// SIMATIC STEP 7 (V5.x) project KROMOSS_RULLIERA_EIDOS
// station: Hardware
// station: SIMATIC 300
// station: P_ADR_BUS
// station: P_ADR_BUS
// station: Configurazione
// program: Programma S7
// program: Backup
// program: MICROMASTER_420
// program: MICROMASTER_420
// program: MICROMASTER_420
// program: MICROMASTER_420
// program: MICROMASTER_420
// program: MICROMASTER_420
// program: MICROMASTER_420
// program: MICROMASTER_420
// program: MICROMASTER_420
// program: MICROMASTER_420
// program: MICROMASTER_420
// program: MICROMASTER_420
// program: MICROMASTER_420
// program: MICROMASTER_420
// program: MICROMASTER_420
// program: MICROMASTER_420

SYMBOL_TABLE
"C1"	C 1	COUNTER	// TIMEOUT TRASFERIMENTO "M3"
"C2"	C 2	COUNTER	// TEMPO SVUOTAMENTO CATENA INGRESSO CADENZATORE LINEA 2
"C3"	C 3	COUNTER	// TEMPO PASSO CATENE LINEA 2
"C4"	C 4	COUNTER	// TEMPO PASSO CATENE ACCUMULO "A" LINEA 2
"C5"	C 5	COUNTER	// TEMPO SVUOTAMENTO CATENA INGRESSO CADENZATORE LINEA 1
"C6"	C 6	COUNTER	// TEMPO PASSO CATENE LINEA 1
"C7"	C 7	COUNTER
"C8"	C 8	COUNTER
"C9"	C 9	COUNTER	// CONTEGGIO PEZZI SU CATENA FISSA LINEA 2
"C10"	C 10	COUNTER
"C11"	C 11	COUNTER
"C12"	C 12	COUNTER
"C13"	C 13	COUNTER	// CONTEGGIO PEZZI SU CATENA FISSA LINEA 1
"C14"	C 14	COUNTER
"C15"	C 15	COUNTER
"C16"	C 16	COUNTER
"C17"	C 17	COUNTER
"C18"	C 18	COUNTER
"C19"	C 19	COUNTER
"C20"	C 20	COUNTER	// RITARDO FUORI INGOMBRO M22
"C21"	C 21	COUNTER	// RITARDO FUORI INGOMBRO M24
"DB_OP"	DB 2	DB 2
"DB_InverterParams"	DB 3	DB 3
"DB_Accumulo"	DB 10	DB 10
"DETAIL_DIAG_DB"	DB 125	FB 125
"DB_ReadParamLoop"	DB 211	FB 211
"DB_GestCodeEstrusori"	DB 212	FB 212
"DB_LinkEthernet_1"	DB 213	FB 213
"DB_LinkEthernet_2"	DB 214	FB 213
"DETAIL_DP_DIAG"	FB 125	FB 125
"ReadParamInverters"	FB 210	FB 210
"FB_ReadParamLoop"	FB 211	FB 211
"FB_GestCodeEstrusori"	FB 212	FB 212
"FB_LinkEthernet"	FB 213	FB 213
"Allarmi"	FC 1	FC 1	// Gestione allarmi
"Segnalazioni"	FC 2	FC 2	// Gestione segnalazioni
"Consensi Generali"	FC 3	FC 3	// Consensi generali
"Automatico_zona_ingresso"	FC 4	FC 4	// Condizioni automatico zona ingresso
"Automatico_linea_1"	FC 5	FC 5	// Condizioni automatico linea 1
"Automatico_linea_2"	FC 6	FC 6	// Condizioni automatico linea 2
"PROFIBUS_MM4"	FC 10	FC 10
"Comandi_zona_ingresso"	FC 14	FC 14	// Comandi utenze zona ingresso
"Comandi_linea_1"	FC 15	FC 15	// Comandi utenze linea 1
"Comandi_linea_2"	FC 16	FC 16	// Comandi utenze linea 2
"Comandi_Inverter"	FC 17	FC 17
"Gestione finecorsa"	FC 18	FC 18
"Gestione OP"	FC 20	FC 20
"Gestione Timer e Counter"	FC 30	FC 30
"AG_SEND"	FC 106	FC 106	// AG SEND
"AG_RECV"	FC 107	FC 107	// AG RECEIVE
"MM4_ReadWrite_Param"	FC 200	FC 200
"FC_AllarmeAttivo"	FC 201	FC 201
"FC_ResetAllarmi"	FC 202	FC 202
"FC_ControlloMsgEth"	FC 203	FC 203
"InvertiMinuscMaiusc"	FC 204	FC 204
"Termico_M1"	I 0.0	BOOL
"Termico_M2"	I 0.1	BOOL
"Termico_M3"	I 0.2	BOOL
"Termico_M4"	I 0.3	BOOL
"Termico_M5"	I 0.4	BOOL
"Termico_M6"	I 0.5	BOOL
"Termico_M7"	I 0.6	BOOL
"Termico_M8"	I 0.7	BOOL
"Termico_M9"	I 1.0	BOOL
"Termico_M10"	I 1.1	BOOL
"Termico_M11"	I 1.2	BOOL
"Termico_M12"	I 1.3	BOOL
"Termico_M13"	I 1.4	BOOL
"Termico_M14"	I 1.5	BOOL
"Termico_M15"	I 1.6	BOOL
"Termico_M16"	I 1.7	BOOL
"Termico_M17"	I 2.0	BOOL
"Termico_M18"	I 2.1	BOOL
"Termico_M19"	I 2.2	BOOL
"Termico_Avviatore_Spare"	I 2.3	BOOL
"Spare_1"	I 2.4	BOOL
"Spare_2"	I 2.5	BOOL
"Spare_3"	I 2.6	BOOL
"Spare_4"	I 2.7	BOOL
"QF20_Inverter_M20"	I 3.0	BOOL
"QF21_Inverter_M21"	I 3.1	BOOL
"QF22_Inverter_M22"	I 3.2	BOOL
"QF23_Inverter_M23"	I 3.3	BOOL
"QF24_Inverter_M24"	I 3.4	BOOL
"QF25_Inverter_M25"	I 3.5	BOOL
"QF26_Inverter_M26"	I 3.6	BOOL
"QF27_Inverter_M27"	I 3.7	BOOL
"QF28_Inverter_M28"	I 4.0	BOOL
"QF29_Inverter_M29"	I 4.1	BOOL
"QF30_Inverter_M30"	I 4.2	BOOL
"QF31_Inverter_M31"	I 4.3	BOOL
"QF32_Inverter_M32"	I 4.4	BOOL
"QF33_Inverter_M33"	I 4.5	BOOL
"QF34_Inverter_M34"	I 4.6	BOOL
"QF35_Inverter_M35"	I 4.7	BOOL
"QF36_Spare"	I 5.0	BOOL
"QF6_Ventilazione_Quadro"	I 5.1	BOOL
"QF8_Alim_PS_Comandi"	I 5.2	BOOL
"QF19_Alim_Circuiti_Emerg"	I 5.3	BOOL
"QF10_Alim_Comandi_Quadro"	I 5.4	BOOL
"QF11_Alim_Comandi_JP1"	I 5.5	BOOL
"QF12_Alim_Comandi_JP2"	I 5.6	BOOL
"QF13_Alim_Comandi_JP3"	I 5.7	BOOL
"PULSANTE_RESET"	I 6.0	BOOL
"Selettore_Spare_2"	I 6.1	BOOL
"Selettore_Abil_Linea1"	I 6.2	BOOL
"Selettore_Abil_Linea2"	I 6.3	BOOL
"Selettore_Abil_Laser"	I 6.4	BOOL
"Selettore_Abil_Stampanti"	I 6.5	BOOL
"Impianto_AUT"	I 6.6	BOOL
"Impianto_MAN"	I 6.7	BOOL
"Proximity_1_pos_laser1"	I 7.0	BOOL
"Proximity_2_ingr_moret1"	I 7.1	BOOL
"Proximity_1_pos_laser2"	I 7.2	BOOL
"Proximity_2_ingr_moret2"	I 7.3	BOOL
"Spare_5"	I 7.4	BOOL
"Spare_6"	I 7.5	BOOL
"Spare_7"	I 7.6	BOOL
"Spare_8"	I 7.7	BOOL
"Spare_9"	I 8.0	BOOL
"Traslatore_Alto_SX"	I 20.0	BOOL
"Traslatore_Basso_SX"	I 20.1	BOOL
"Traslatore_Alto_DX"	I 20.2	BOOL
"Traslatore_Basso_DX"	I 20.3	BOOL
"IR_Stop_Traslazione"	I 20.4	BOOL
"Stop_Profili_OUT_Impiant"	I 20.5	BOOL
"Nastro_Deposito1_Alto_DX"	I 21.0	BOOL
"Nastro_Deposito1_Bass_DX"	I 21.1	BOOL
"Nastro_Deposito1_Alto_SX"	I 21.2	BOOL
"Nastro_Deposito1_Bass_SX"	I 21.3	BOOL
"Nastro_Prelievo1_Alto_SX"	I 21.4	BOOL
"Nastro_Prelievo1_Bass_SX"	I 21.5	BOOL
"Nastro_Prelievo1_Alto_DX"	I 21.6	BOOL
"Nastro_Prelievo1_Bass_DX"	I 21.7	BOOL
"Nastro_Prelievo2_Alto_DX"	I 22.0	BOOL
"Nastro_Prelievo2_Bass_DX"	I 22.1	BOOL
"Nastro_Prelievo2_Alto_SX"	I 22.2	BOOL
"Nastro_Prelievo2_Bass_SX"	I 22.3	BOOL
"Nastro_Deposito2_Alto_DX"	I 22.4	BOOL
"Nastro_Deposito2_Bass_DX"	I 22.5	BOOL
"Nastro_Deposito2_Alto_SX"	I 22.6	BOOL
"Nastro_Deposito2_Bass_SX"	I 22.7	BOOL
"IR_Stop_Nastro_Scarico1"	I 23.0	BOOL
"IR_Stop_Barra_accumulo2"	I 23.1	BOOL
"IR_Stop_Nastro_Prelievo1"	I 23.2	BOOL
"IR_Stop_Nastro_Prelievo2"	I 23.3	BOOL
"IR_Stop_Barra_accumulo1"	I 23.4	BOOL
"IR_Stop_Nastro_Scarico2"	I 23.5	BOOL
"FTC_Stop_4profili_prel_1"	I 23.6	BOOL
"FTC_Stop_4profili_prel_2"	I 23.7	BOOL
"Proximity_0_Cadenzatore1"	I 24.0	BOOL
"Proximity_0_Cadenzatore2"	I 24.1	BOOL
"Nastro_Scarico1_Alto_DX"	I 25.0	BOOL
"Nastro_Scarico1_Bass_DX"	I 25.1	BOOL
"Nastro_Scarico1_Alto_SX"	I 25.2	BOOL
"Nastro_Scarico1_Bass_SX"	I 25.3	BOOL
"Nastro_Scarico2_Alto_DX"	I 25.4	BOOL
"Nastro_Scarico2_Bass_DX"	I 25.5	BOOL
"Nastro_Scarico2_Alto_SX"	I 25.6	BOOL
"Nastro_Scarico2_Bass_SX"	I 25.7	BOOL
"IR_Start_Banco1_Scaric_L"	I 26.0	BOOL
"IR_Stop_Banco1_Scaric_L"	I 26.1	BOOL
"IR_Start_Banco2_Scaric_L"	I 26.2	BOOL
"IR_Stop_Banco2_Scaric_L"	I 26.3	BOOL
"IR_Stop_Banco1_Scaric_H"	I 26.4	BOOL
"IR_Stop_Banco2_Scaric_H"	I 26.5	BOOL
"FTC_Stop_rull1_out_ext"	I 26.6	BOOL
"FTC_Stop_rull2_out_ext"	I 26.7	BOOL
"FTC_Stop_rull1_out_int"	I 27.0	BOOL
"FTC_Stop_rull2_out_int"	I 27.1	BOOL
"Proximity_0_Cadenz_scar1"	I 27.2	BOOL
"Proximity_0_Cadenz_scar2"	I 27.3	BOOL
"I96.0"	I 96.0	BOOL	// CONSENSO DA FORNO PER RULLIERE
"OFF"	M 0.0	BOOL
"ON"	M 0.1	BOOL
"TODO"	M 0.2	BOOL
"BYPASS"	M 0.3	BOOL
"MANUALE"	M 1.0	BOOL	// IMPIANTO IN MANUALE
"AUTOMATICO"	M 1.1	BOOL	// IMPIANTO IN AUTOMATICO
"AUTO_LINEA_1"	M 1.2	BOOL	// LINEA 1 INSERITA E IN AUTOMATICO
"AUTO_LINEA_2"	M 1.3	BOOL	// LINEA 2 INSERITA E IN AUTOMATICO
"AUTO_LASER"	M 1.4	BOOL	// LASER INSERITO E IN AUTOMATICO
"AUTO_STAMPA"	M 1.5	BOOL	// STAMPANTE INSERITA E IN AUTOMATICO
"EMERGENZA"	M 1.6	BOOL	// IMPIANTO IN EMERGENZA
"ALLARME"	M 1.7	BOOL	// ALMENO UN ALLARME ATTIVO
"PULSE_AUTOMATICO"	M 2.0	BOOL
"PULSE_MANUALE"	M 2.1	BOOL
"M3.0"	M 3.0	BOOL	// ALMENO UN ALLARME ATTIVO
"occhio"	M 4.0	BOOL
"M2_Presenza"	M 10.0	BOOL	// PACCO IN POSIZIONE PER TRASFERIMENTO CON "M3"
"M10.1"	M 10.1	BOOL	// MEM AUITO SALITA TRASLATORE "M3"
"M10.2"	M 10.2	BOOL	// MEM AUTO MARCIA TRASLATORE "M3"
"M10.3"	M 10.3	BOOL	// CONSENSO DISCESA TRASLATORE "M3"
"M20_Presenza"	M 11.0	BOOL	// PACCO IN POSIZIONE SU RULLIERA 1 A 4 FILE
"M11.1"	M 11.1	BOOL	// TRASFERISCI PACCO 4 FILE SU LINEA 2
"M11.2"	M 11.2	BOOL	// TRASFERISCI RULLI 4 FILE SU LINEA 1
"M11.3"	M 11.3	BOOL	// MEM AUTO RULLI "M20"
"M11.4"	M 11.4	BOOL	// MEM AUTO RULLI "M21"
"M11.5"	M 11.5	BOOL	// MEM AUTO RULLI "M22"
"M11.6"	M 11.6	BOOL	// MEM AUTO RULLI "M23"
"M11.7"	M 11.7	BOOL	// MEM AUTO RULLI "M24"
"M20.0"	M 20.0	BOOL	// CONSENSO START CADENZATORE "M7"
"M20.1"	M 20.1	BOOL	// PRENOTA TRASFERIMENTO SU LINEA 2
"M20.2"	M 20.2	BOOL	// CONSENSO TRASFERIMENTO PACCO 4 FILE SU LINEA 2
"M22_Presenza"	M 20.3	BOOL	// PACCO 4 FILE IN POSIZIONE DAVANTI LINEA 2
"M20.4"	M 20.4	BOOL	// MEM AUTO SOLLEVA CATENA INGRESSO LINEA 2
"M20.5"	M 20.5	BOOL	// MEM AUTO CATENE INGRESSO LINEA 2 "M4"
"M20.6"	M 20.6	BOOL	// MEM AUTO ABBASSA CATENE INGRESSO LINEA 2
"M20.7"	M 20.7	BOOL	// MEM PRENOTA CICLO CADENZATORE LINEA 2
"M21.0"	M 21.0	BOOL	// MEM AUTO PACCO IN INGRESSO CADEZ. LINEA 2
"M21.1"	M 21.1	BOOL	// MEM AUTO CICLO CADENZATORE LINEA 2
"M21.2"	M 21.2	BOOL	// CICLO CADENZATORE IN CORSO LINEA 2
"M21.3"	M 21.3	BOOL	// LINEA 2 FAI PASSO CATENE
"M21.4"	M 21.4	BOOL	// MEM AUTO CATENA "M5"
"M21.5"	M 21.5	BOOL	// MEM AUTO CATENA "M6"
"M21.6"	M 21.6	BOOL	// FINE CICLO CADENZATORE LINEA 2
"M22.0"	M 22.0	BOOL	// PROFILATO IN USCITA CATENA CADEZ. LINEA 2
"M22.1"	M 22.1	BOOL	// PROFILATO SU RULLIERA 1 INGRESSO ESTR. LINEA 2
"M22.2"	M 22.2	BOOL	// MEM PROFILATO SU RULLIERA 2 LINEA 2
"M22.3"	M 22.3	BOOL	// RULLIERA 1 INGRESSO ESTR. LINEA 2 LIBERA
"M22.4"	M 22.4	BOOL	// MEM AUTO SOLLEVA CATENA USCITA CADEZ. LINEA 2
"M22.5"	M 22.5	BOOL	// MEM AUTO ABBASSA CATENA USCITA CADEZ. LINEA 2
"M22.6"	M 22.6	BOOL	// MEM AUTO RULLIERA 1 INGRESSO ESTR. LINEA 2 "M25"
"M22.7"	M 22.7	BOOL	// MEM AUTO RULLIERA 2 INGRESSO ESTR. LINEA 2 "M26"
"M23.0"	M 23.0	BOOL	// MEM MANUALE CADENZ. "A" LINEA 2
"M23.7"	M 23.7	BOOL	// RICHIEDI CONFERMA TIPO BARRA SU LINEA 2
"M24.0"	M 24.0	BOOL	// PRONTATO SCARICO ACCUMULO "A" LINEA 2
"M24.1"	M 24.1	BOOL	// PRENOTA CICLO CADEZ. "A" LINEA 2
"M24.2"	M 24.2	BOOL	// MEM AUTO CICLO CADEZ. "A" LINEA 2
"M24.3"	M 24.3	BOOL	// CICLO CADEZ. "A" LINEA 2 IN CORSO
"M24.4"	M 24.4	BOOL	// CICLO CADENZATORE TERMINATO LINEA 2
"M24.5"	M 24.5	BOOL	// MEM AUTO RULLIERA "M30"
"M24.6"	M 24.6	BOOL	// PASSO CATENA ACCUMULO LINEA "A"
"M24.7"	M 24.7	BOOL	// MEM AUTO CATENE "M17"
"M25.0"	M 25.0	BOOL	// TRASFERISCI PACCO CADENZATO IN USCITA
"M25.1"	M 25.1	BOOL	// BARRA DA SCARICARE SU ACCUMULO "B"
"M25.2"	M 25.2	BOOL	// SPOSTA BARRA RU RULLIERA "M31"
"M25.3"	M 25.3	BOOL	// MEM AUTO RULLIERA "M31"
"M25.4"	M 25.4	BOOL	// PRENOTA CICLO CADENZATORE "B"
"M25.5"	M 25.5	BOOL	// MEM AUTO CICLO CADENZ. "B" LINEA 2
"M25.6"	M 25.6	BOOL	// CICLO CADEZ. "B2 IN CORSO
"M25.7"	M 25.7	BOOL	// CICLO CADENZATORE "B" TERMINATO
"M26.0"	M 26.0	BOOL	// MEM MANUALE CADENZ. "B" LINEA 2
"Avvio_M30_L2"	M 26.2	BOOL
"M26.4"	M 26.4	BOOL	// PASSO CATENA ACCULULO "B"
"M26.7"	M 26.7	BOOL	// MEM AUTO CATENE "M19"
"Attesa Conferma Scarico2"	M 27.0	BOOL
"M40.0"	M 40.0	BOOL	// CONSENSO START CADENZATORE "M8"
"M40.1"	M 40.1	BOOL	// PRENOTA TRASFERIMENTO SU LINEA 1
"M40.2"	M 40.2	BOOL	// CONSENSO TRASFERIMENTO 4 FILE SU LINEA 1
"M24_Presenza"	M 40.3	BOOL	// PACCO 4 FILE IN POSIZIONE DAVANTI LINEA 1
"M40.4"	M 40.4	BOOL	// MEM AUTO SOLLEVA CATENA INGRESSO LINEA 1
"M40.5"	M 40.5	BOOL	// MEM AUTO CATENE INGRESSO LINEA 1 "M11"
"M40.6"	M 40.6	BOOL	// MEM AUTO ABBASSA CATENE INGRESSO LINEA 1
"M40.7"	M 40.7	BOOL	// MEM PRENOTA CICLO CADENZATORE LINEA 1
"M41.0"	M 41.0	BOOL	// MEM AUTO PACCO IN INGRESSO CADEZ. LINEA 1
"M41.1"	M 41.1	BOOL	// MEM AUTO PACCO IN INGRESSO CADENZ. LINEA 1 "M8"
"M41.2"	M 41.2	BOOL	// CICLO CADENZATORE IN CORSO LINEA 1
"M41.3"	M 41.3	BOOL	// CICLO CADENZATORE TERMINATO LINEA 1
"M41.4"	M 41.4	BOOL	// MEM AUTO CATENA "M10"
"M41.5"	M 41.5	BOOL	// MEM AUTO CATENA "M9"
"M41.6"	M 41.6	BOOL	// FINE CICLO CADENZATORE LINEA 1
"M42.0"	M 42.0	BOOL	// PROFILATO IN USCITA CATENA CADEZ. LINEA 1
"M27_Presenza"	M 42.1	BOOL	// PROFILATO SU RULLIERA 1 INGRESSO ESTR. LINEA 1
"M42.2"	M 42.2	BOOL	// MEM PROFILATO SU RULLIERA 2 LINEA 1
"M42.3"	M 42.3	BOOL	// RULLIERA 1 INGRESSO ESTR. LINEA 2 LIBERA
"M42.4"	M 42.4	BOOL	// MEM AUTO SOLLEVA CATENA USCITA CADENZ. LINEA 1
"M42.5"	M 42.5	BOOL	// MEM AUTO ABBASSA CATENA USCITA CADENZ. LINEA 1
"M42.6"	M 42.6	BOOL	// MEM AUTO RULLIERA 1 INGRESSO ESTR. LINEA 1 "M27"
"M42.7"	M 42.7	BOOL	// MEM AUTO RULLIERA 2 INGRESSO ESTR. LINEA 1 "M28"
"M43.0"	M 43.0	BOOL	// MEM AUTO RULLIERA 3 INGRESSO ESTR. LINEA 1 "M29"
"M43.1"	M 43.1	BOOL	// PROFILATO IN USCITA DA ESTRUSORE 1
"M43.2"	M 43.2	BOOL	// MEM AUTO RULLI "M32"
"M43.3"	M 43.3	BOOL	// MEM AUTO RULLI "M33"
"M43.4"	M 43.4	BOOL	// MEM AUTO RULLI "M34"
"M43.5"	M 43.5	BOOL	// CATENA SVINCOLO "A" LINEA 1 ALTA
"M43.6"	M 43.6	BOOL	// CATENA SVINCOLO "A" LINEA 1 BASSA
"M43.7"	M 43.7	BOOL	// RICHIEDI CONFERMA TIPO BARRA SU LINEA 1
"M44.0"	M 44.0	BOOL	// PRENOTA SCARICO SU "A" LINEA 1
"M44.1"	M 44.1	BOOL	// CARICA SU SCARICO "A" LINEA 1
"M44.2"	M 44.2	BOOL	// MEM AUTO SOLLEVA CATENE SVINCOLO "A" LINEA 1
"M44.3"	M 44.3	BOOL	// MEM AUTO ABBASSA CATENE SVINCOLO "A" LINEA 1
"M44.4"	M 44.4	BOOL	// MEM AUTO CATENE ACCUMULO "A" LINEA 1 "M12"
"M44.5"	M 44.5	BOOL	// MEM AUTO CATENE ACCUMULO "A" LINEA 1 "M13"
"M45.0"	M 45.0	BOOL	// TRASFERISCI PACCO CADENZATO IN USCITA
"M45.1"	M 45.1	BOOL	// BARRA DA SCARICARE SU ACCUMULO "B"
"M45.2"	M 45.2	BOOL	// SPOSTA BARRA SU RULLIERA "M34"
"M45.4"	M 45.4	BOOL	// MEM CICLO DEVIAZIONE ACCUMULO "B"
"M45.5"	M 45.5	BOOL	// MEM AUTO ALZA CATENE SVINCOLO "B" LINEA 1
"M45.6"	M 45.6	BOOL	// MEM AUTO ABBASSA CATENE SVINCOLO "B" LINEA 1
"M46.0"	M 46.0	BOOL	// MEM AUTO CATENE ACCUMULO "B" LINEA 1 "M14"
"M46.1"	M 46.1	BOOL	// MEM AUTO CATENE ACCUMULO "B" LINEA 1 "M15"
"Attesa Conferma Scarico1"	M 47.0	BOOL
"Comando_M20"	M 64.0	BOOL	// Motore rulliera 4 profili pos.1
"Comando_M21"	M 64.1	BOOL	// Motore rulliera 4 profili pos.2
"Comando_M22"	M 64.2	BOOL	// Motore rulliera 4 profili pos.3
"Comando_M23"	M 64.3	BOOL	// Motore rulliera 4 profili pos.4
"Comando_M24"	M 64.4	BOOL	// Motore rulliera 4 profili pos.5
"Comando_M25"	M 64.5	BOOL	// Motore rulliera ingresso S1-1
"Comando_M26"	M 64.6	BOOL	// Motore rulliera ingresso S1-2
"Comando_M27"	M 64.7	BOOL	// Motore rulliera ingresso S2-1
"Comando_M28"	M 65.0	BOOL	// Motore rulliera ingresso S2-2
"Comando_M29"	M 65.1	BOOL	// Motore rulliera ingresso S2-3
"Comando_M30"	M 65.2	BOOL	// Motore rulliera uscita S1-3
"Comando_M31"	M 65.3	BOOL	// Motore rulliera uscita S1-4
"Comando_M32"	M 65.4	BOOL	// Motore rulliera uscita S2-4
"Comando_M33"	M 65.5	BOOL	// Motore rulliera uscita S2-5
"Comando_M34"	M 65.6	BOOL	// Motore rulliera uscita S2-6
"Comando_M35"	M 65.7	BOOL	// Motore rulliera uscita S2-7
"M66.0"	M 66.0	BOOL	// INVERTER A1 FAULT
"M66.1"	M 66.1	BOOL	// INVERTER A2 FAULT
"M66.2"	M 66.2	BOOL	// INVERTER A3 FAULT
"M66.3"	M 66.3	BOOL	// INVERTER A4 FAULT
"M66.4"	M 66.4	BOOL	// INVERTER A5 FAULT
"M66.5"	M 66.5	BOOL	// INVERTER A6 FAULT
"M66.6"	M 66.6	BOOL	// INVERTER A7 FAULT
"M66.7"	M 66.7	BOOL	// INVERTER A8 FAULT
"M67.0"	M 67.0	BOOL	// INVERTER A9 FAULT
"M67.1"	M 67.1	BOOL	// INVERTER A10 FAULT
"M67.2"	M 67.2	BOOL	// INVERTER A11 FAULT
"M67.3"	M 67.3	BOOL	// INVERTER A12 FAULT
"M67.4"	M 67.4	BOOL	// INVERTER A13 FAULT
"M67.5"	M 67.5	BOOL	// INVERTER A14 FAULT
"M67.6"	M 67.6	BOOL	// INVERTER A15 FAULT
"M67.7"	M 67.7	BOOL	// INVERTER A16 FAULT
"M68.0"	M 68.0	BOOL	// MEM AUTOMATICO M1/M2 PROVVISORIO
"M70.0"	M 70.0	BOOL	// MOTORE M1 IN ALLARME
"M70.1"	M 70.1	BOOL	// MOTORE M2 IN ALLARME
"M70.2"	M 70.2	BOOL	// MOTORE M3 IN ALLARME
"M70.3"	M 70.3	BOOL	// MOTORE M4 IN ALLARME
"M70.4"	M 70.4	BOOL	// MOTORE M5 IN ALLARME
"M70.5"	M 70.5	BOOL	// MOTORE M6 IN ALLARME
"M70.6"	M 70.6	BOOL	// MOTORE M7 IN ALLARME
"M70.7"	M 70.7	BOOL	// MOTORE M8 IN ALLARME
"M71.0"	M 71.0	BOOL	// MOTORE M9 IN ALLARME
"M71.1"	M 71.1	BOOL	// MOTORE M10 IN ALLARME
"M71.2"	M 71.2	BOOL	// MOTORE M11 IN ALLARME
"M71.3"	M 71.3	BOOL	// MOTORE M12 IN ALLARME
"M71.4"	M 71.4	BOOL	// MOTORE M13 IN ALLARME
"M71.5"	M 71.5	BOOL	// MOTORE M14 IN ALLARME
"M71.6"	M 71.6	BOOL	// MOTORE M15 IN ALLARME
"M71.7"	M 71.7	BOOL	// MOTORE M16 IN ALLARME
"M72.0"	M 72.0	BOOL	// MOTORE M17 IN ALLARME
"M72.1"	M 72.1	BOOL	// MOTORE M18 IN ALLARME
"M72.2"	M 72.2	BOOL	// MOTORE M19 IN ALLARME
"M72.3"	M 72.3	BOOL	// MOTORE M20 IN ALLARME
"M72.4"	M 72.4	BOOL	// MOTORE M21 IN ALLARME
"M72.5"	M 72.5	BOOL	// MOTORE M22 IN ALLARME
"M72.6"	M 72.6	BOOL	// MOTORE M23 IN ALLARME
"M72.7"	M 72.7	BOOL	// MOTORE M24 IN ALLARME
"M73.0"	M 73.0	BOOL	// MOTORE M25 IN ALLARME
"M73.1"	M 73.1	BOOL	// MOTORE M26 IN ALLARME
"M73.2"	M 73.2	BOOL	// MOTORE M27 IN ALLARME
"M73.3"	M 73.3	BOOL	// MOTORE M28 IN ALLARME
"M73.4"	M 73.4	BOOL	// MOTORE M29 IN ALLARME
"M73.5"	M 73.5	BOOL	// MOTORE M30 IN ALLARME
"M73.6"	M 73.6	BOOL	// MOTORE M31 IN ALLARME
"M73.7"	M 73.7	BOOL	// MOTORE M32 IN ALLARME
"M74.0"	M 74.0	BOOL	// MOTORE M33 IN ALLARME
"M74.1"	M 74.1	BOOL	// MOTORE M34 IN ALLARME
"M74.2"	M 74.2	BOOL	// MOTORE M35 IN ALLARME
"M74.3"	M 74.3	BOOL	// NODO JP1 ET200S OK
"M74.4"	M 74.4	BOOL	// NODO JP2 ET200S OK
"M74.5"	M 74.5	BOOL	// NODO JP3 ET200S OK
"M80.0"	M 80.0	BOOL	// AUX PULSE 1
"M80.1"	M 80.1	BOOL	// AUX PULSE 2
"M80.2"	M 80.2	BOOL	// AUX PULSE 3
"M80.3"	M 80.3	BOOL	// AUX PULSE 4
"M80.4"	M 80.4	BOOL	// AUX PULSE
"M80.5"	M 80.5	BOOL	// AUX PULSE
"M80.6"	M 80.6	BOOL	// AUX PULSE
"M80.7"	M 80.7	BOOL	// AUX PULSE
"M81.0"	M 81.0	BOOL	// AUX PULSE
"M81.1"	M 81.1	BOOL	// AUX PULSE
"M81.2"	M 81.2	BOOL	// AUX PULSE
"M81.3"	M 81.3	BOOL	// AUX PULSE
"M81.4"	M 81.4	BOOL	// AUX PULSE
"M81.5"	M 81.5	BOOL	// AUX PULSE
"M81.6"	M 81.6	BOOL
"M81.7"	M 81.7	BOOL
"M82.0"	M 82.0	BOOL
"M82.1"	M 82.1	BOOL
"M82.2"	M 82.2	BOOL	// AUX PULSE
"M82.3"	M 82.3	BOOL	// AUX PULSE
"M82.4"	M 82.4	BOOL	// AUX PULSE
"M90.0"	M 90.0	BOOL	// AUX START MANUALE "M7"
"M90.1"	M 90.1	BOOL	// PULSE STOP CADENZATORE "M7"
"M90.2"	M 90.2	BOOL	// AUX START MANUALE "M8"
"M90.3"	M 90.3	BOOL	// PULSE STOP CADENZATORE "M8"
"M90.4"	M 90.4	BOOL	// START MANUALE CADEZ. "A" LINEA 2
"M90.5"	M 90.5	BOOL	// STOP FASE CADEZ. "A" LINEA 2
"M90.6"	M 90.6	BOOL	// START MANUALE CADEZ. "B" LINEA 2
"M90.7"	M 90.7	BOOL	// STOP FASE CADEZ. "B" LINEA 2
"M99.0"	M 99.0	BOOL
"M99.1"	M 99.1	BOOL
"M99.2"	M 99.2	BOOL
"M99.3"	M 99.3	BOOL
"M100.0"	M 100.0	BOOL	// PAGINE ATTIVE: MANUALE
"M100.1"	M 100.1	BOOL	// PAGINE ATTIVE: AUTOMATICO
"M100.2"	M 100.2	BOOL	// PAGINE ATTIVE: DIAGNOSTICA PROFIBUS
"M100.3"	M 100.3	BOOL	// FORZA CAMBIO PAGINA
"M100.4"	M 100.4	BOOL	// PAGINA ATTIVA: EMERGENZA
"M100.5"	M 100.5	BOOL	// PAGINA ATTIVA: MACCHINA SPENTA
"M100.6"	M 100.6	BOOL	// PAGINE ATTIVE: STATO
"M100.7"	M 100.7	BOOL	// RICHIEDI CAMBIO PAGINA
"NewStrEthLinea1"	M 101.0	BOOL	// NUOVO MESSAGGIO ETH SU PORT 2000
"Linea1Str_L1"	M 101.1	BOOL	// RICEVUTO "L1" SU PORT 2000
"Linea1Str_L2"	M 101.2	BOOL	// RICEVUTO "L2" SU PORT 2000
"LinkEth1_Ok"	M 101.3	BOOL	// COLLEGAMENTO ETH PROT 2000 OK
"LinkEth1_Error"	M 101.4	BOOL	// COLLEGAMENTO ETH PROT 2000 KO
"NewStrEthLinea2"	M 102.0	BOOL	// NUOVO MESSAGGIO ETH SU PORT 2001
"Linea2Str_L1"	M 102.1	BOOL	// RICEVUTO "L1" SU PORT 2001
"Linea2Str_L2"	M 102.2	BOOL	// RICEVUTO "L2" SU PORT 2001
"LinkEth2_Ok"	M 102.3	BOOL	// COLLEGAMENTO ETH PROT 2001 OK
"LinkEth2_Error"	M 102.4	BOOL	// COLLEGAMENTO ETH PROT 2001 KO
"ByPass1ConfermadaPannell"	M 103.0	BOOL
"M103.1"	M 103.1	BOOL
"ByPass2ConfermadaPannell"	M 103.2	BOOL
"M103.3"	M 103.3	BOOL
"M120.0"	M 120.0	BOOL	// TRASLATORE "M3" ALTO
"M120.1"	M 120.1	BOOL	// TRASLATORE "M3" BASSO
"M120.2"	M 120.2	BOOL	// NASTRO PRELIEVO LINEA 2 ALTO
"M120.3"	M 120.3	BOOL	// NASTRO PRELIEVO LINEA 2 BASSO
"M120.4"	M 120.4	BOOL	// CATENA INGRESSO CAD. LINEA 2 SVUOTATA
"M120.5"	M 120.5	BOOL	// TEMPO PASSO CATENE LINEA 2
"M120.6"	M 120.6	BOOL	// NASTRO USCITA CAD. LINEA 2 ALTO
"M120.7"	M 120.7	BOOL	// NASTRO USCITA CAD. LINEA 2 BASSO
"M121.0"	M 121.0	BOOL	// TEMPO PASSO CATENE ACCUMULO "A" LINEA 2
"M121.1"	M 121.1	BOOL	// NASTRO PRELIEVO LINEA 1 ALTO
"M121.2"	M 121.2	BOOL	// NASTRO PRELIEVO LINEA 1 BASSO
"M121.3"	M 121.3	BOOL	// CATENA INGRESSO CAD. LINEA 1 SVUOTATA
"M121.4"	M 121.4	BOOL	// TEMPO PASSO CATENE LIINEA 1
"M121.5"	M 121.5	BOOL	// NASTRO USCITA CAD. LINEA 1 ALTO
"M121.6"	M 121.6	BOOL	// NASTRO USCITA CAD. LINEA 1 BASSO
"M121.7"	M 121.7	BOOL	// CADENZATORE INGRESSO LINEA 2 FUORI INGOMBRO
"M122.0"	M 122.0	BOOL	// CADENZATORE INGRESSO LINEA 1 FUORI INGOMBRO
"M122.1"	M 122.1	BOOL	// LIMITE PEZZI SU CATENA CADENZATORE LINEA 2
"M122.2"	M 122.2	BOOL	// CATENA USCITA LINEA 2 VUOTA
"M122.3"	M 122.3	BOOL	// CATENA SCARICO LINEA 2 VUOTA
"M122.4"	M 122.4	BOOL	// PACCO IN POSIZIONE SU CATENA USCITA LINEA 2
"M122.5"	M 122.5	BOOL	// RITARDO FUORI INGOMBRO PACCO SU M22
"M122.6"	M 122.6	BOOL	// RITARDO FUORI INGOBRO M24
"M123.1"	M 123.1	BOOL	// LIMITE PEZZI SU CATENA CADENZATORE LINEA 1
"M123.2"	M 123.2	BOOL	// CATENA USCITA LINEA 1 VUOTA
"M123.3"	M 123.3	BOOL	// CATENA SCARICO LINEA 1 VUOTA
"M123.4"	M 123.4	BOOL	// PACCO IN POSIZIONE SU CATENA USCITA LINEA 1
"M123.5"	M 123.5	BOOL	// PASSO CATENA ACCUMULO "A" LINEA 1
"M123.6"	M 123.6	BOOL	// TEMPO PASSO CATENE LINEA 2 "B"
"M123.7"	M 123.7	BOOL	// PASSO CATENA ACCUMULO "B" LINEA 1
"M130.0"	M 130.0	BOOL	// MEM FC TRASLATORE INGRESSO ALTO
"M130.1"	M 130.1	BOOL	// MEM FC TRASLATORE INGRESSO BASSO
"M130.2"	M 130.2	BOOL	// MEM FC CATENE INGRESSO LINEA 2 ALTE
"M130.3"	M 130.3	BOOL	// MEM FC CATENE INGRESSO LINEA 2 BASSE
"M130.4"	M 130.4	BOOL	// MEM FC CATENE USCITA LINEA 2 ALTE
"M130.5"	M 130.5	BOOL	// MEM FC CATENE USCITA LINEA 2 BASSE
"M130.6"	M 130.6	BOOL	// MEM FC CATENE INGRESSO LINEA 1 ALTE
"M130.7"	M 130.7	BOOL	// MEM FC CATENE INGRESSO LINEA 1 BASSE
"M131.0"	M 131.0	BOOL	// MEM FC CATENE USCITA LINEA 1 ALTE
"M131.1"	M 131.1	BOOL	// MEM FC CATENE USCITA LINEA 1 BASSE
"M131.2"	M 131.2	BOOL	// MEM FC CATENE ACCULULO "A" LINEA 1 ALTE
"M131.3"	M 131.3	BOOL	// MEM FC CATENE ACCULULO "A" LINEA 1 BASSE
"M131.4"	M 131.4	BOOL	// MEM FC CATENE ACCULULO "B" LINEA 1 ALTE
"M131.5"	M 131.5	BOOL	// MEM FC CATENE ACCULULO "B" LINEA 1 BASSE
"Linea1_InsCoda"	M 140.0	BOOL
"Linea1_DelCoda"	M 140.1	BOOL
"Linea2_InsCoda"	M 150.0	BOOL
"Linea2_DelCoda"	M 150.1	BOOL
"Mem10Hz"	M 253.0	BOOL
"Mem5Hz"	M 253.1	BOOL
"Mem2,5Hz"	M 253.2	BOOL
"Mem2Hz"	M 253.3	BOOL
"Mem1,25Hz"	M 253.4	BOOL
"Mem1Hz"	M 253.5	BOOL
"Mem0,625Hz"	M 253.6	BOOL
"Mem0,5Hz"	M 253.7	BOOL
"Imp10Hz"	M 254.0	BOOL
"Imp5Hz"	M 254.1	BOOL
"Imp2,5Hz"	M 254.2	BOOL
"Imp2Hz"	M 254.3	BOOL
"Imp1,25Hz"	M 254.4	BOOL
"Imp1Hz"	M 254.5	BOOL
"Imp0,625Hz"	M 254.6	BOOL
"Imp0,5Hz"	M 254.7	BOOL
"10Hz"	M 255.0	BOOL
"5Hz"	M 255.1	BOOL
"2,5Hz"	M 255.2	BOOL
"2Hz"	M 255.3	BOOL
"1,25Hz"	M 255.4	BOOL
"1Hz"	M 255.5	BOOL
"0,625Hz"	M 255.6	BOOL
"0,5Hz"	M 255.7	BOOL
"M280.0"	M 280.0	BOOL	// INCLUDI SCARICO AUTOMATICO
"MemClockBits"	MB 253	BYTE
"ImpClockBits"	MB 254	BYTE
"ClockBits"	MB 255	BYTE
"Linea1_CodiceIn"	MW 142	INT
"Linea1_CodiceOut"	MW 144	INT
"Linea1_ContCoda"	MW 146	INT
"Linea2_CodiceIn"	MW 152	INT
"Linea2_CodiceOut"	MW 154	INT
"Linea2_ContCoda"	MW 156	INT
"CYCL_FLT"	OB 80	OB 80	// Cycle Time Fault
"I/O_FLT1"	OB 82	OB 82	// I/O Point Fault 1
"OBNL_FLT"	OB 85	OB 85	// OB Not Loaded Fault
"RACK_FLT"	OB 86	OB 86	// Loss of Rack Fault
"COMM_FLT"	OB 87	OB 87	// Communication Fault
"COMPLETE RESTART"	OB 100	OB 100	// Complete Restart
"PROG_ERR"	OB 121	OB 121	// Programming Error
"MOD_ERR"	OB 122	OB 122	// Module Access Error
"Comando_M1"	Q 0.0	BOOL	// Motore rulliera 1 estrattore EIDOS
"Comando_M2"	Q 0.1	BOOL	// Motore rulliera 2 estrattore EIDOS
"Comando_M3"	Q 0.2	BOOL	// Motore catena traslazione campata
"Comando_M4"	Q 0.3	BOOL	// Motore catena basculante P1
"Comando_M5"	Q 0.4	BOOL	// Motore catena fissa P1
"Comando_M6"	Q 0.5	BOOL	// Motore catena basculante S1
"Comando_M7"	Q 0.6	BOOL	// Motore cadenzatore P1
"Comando_M8"	Q 0.7	BOOL	// Motore cadenzatore P2
"Comando_M9"	Q 1.0	BOOL	// Motore catena basculante S2
"Comando_M10"	Q 1.1	BOOL	// Motore catena fissa P2
"Comando_M11"	Q 1.2	BOOL	// Motore catena basculante P2
"Comando_M12"	Q 1.3	BOOL	// Motore catena basculante 1
"Comando_M13"	Q 1.4	BOOL	// Motore catena scarico inferiore 1
"Comando_M14"	Q 1.5	BOOL	// Motore catena basculate scarico 2
"Comando_M15"	Q 1.6	BOOL	// Motore catena scarico inferiore 2
"Comando_M16"	Q 1.7	BOOL	// Motore cadenzatore scarico 1
"Comando_M17"	Q 2.0	BOOL	// Motore catena scarico superire 1
"Comando_M18"	Q 2.1	BOOL	// Motore cadenzatore scarico 2
"Comando_M19"	Q 2.2	BOOL	// Motore catena scarico superire 2
"Comando_Spare"	Q 2.3	BOOL
"Comando_KM1_Inverter"	Q 2.7	BOOL
"Gemma_Linea_1"	Q 3.0	BOOL	// SEGNALAZIONE LUMINOSA LINEA 1
"Gemma_Linea_2"	Q 3.1	BOOL	// SEGNALAZIONE LUMINOSA LINEA 2
"Comando_Sirena"	Q 3.2	BOOL
"EV_Chiusura_Allineatori"	Q 3.3	BOOL	// Chiusura allineatori
"Comando_Gemma_Linea2_on"	Q 3.4	BOOL	// LAMPADA VERDE
"Q3.5"	Q 3.5	BOOL	// SEGNALE LUMINOSO ROSSO
"EV_Salita_Traslatore"	Q 20.0	BOOL
"EV_Discesa_Traslatore"	Q 20.1	BOOL
"EV_Salita_Nastro_Depos_1"	Q 21.0	BOOL	// Salita nastro deposito 1
"EV_Discesa_Nastro_Depos1"	Q 21.1	BOOL	// Discesa nastro deposito 1
"EV_Salita_Nastro_Prel_1"	Q 21.2	BOOL	// Salita nastro prelievo 1
"EV_Discesa_Nastro_Prel_1"	Q 21.3	BOOL	// Discesa nastro prelievo 1
"EV_Salita_Nastro_Prel_2"	Q 21.4	BOOL	// Salita nastro deposito 2
"EV_Discesa_Nastro_Prel_2"	Q 21.5	BOOL	// Discesa nastro deposito 2
"EV_Salita_Nastro_Depos_2"	Q 21.6	BOOL	// Salita nastro deposito 2
"EV_Discesa_Nastro_Depos2"	Q 21.7	BOOL	// Discesa nastro deposito 2
"EV_Salita_Nast_Prel_sca1"	Q 23.0	BOOL
"EV_Disce_Nast_Prel_sca1"	Q 23.1	BOOL
"EV_Salita_Nast_Prel_sca2"	Q 23.2	BOOL
"EV_Disce_Nast_Prel_sca2"	Q 23.3	BOOL
"TON"	SFB 4	SFB 4	// Generate an On Delay
"GADR_LGC"	SFC 5	SFC 5	// Query Logical Address of a Channel
"RD_SINFO"	SFC 6	SFC 6	// Read OB Start Information
"D_ACT_DP"	SFC 12	SFC 12	// Deactivating and Activating DP Slaves
"DPNRM_DG"	SFC 13	SFC 13	// Read Diagnostic Data of a DP Slave
"DPRD_DAT"	SFC 14	SFC 14	// Read Consistent Data of a Standard DP Slave
"DPWR_DAT"	SFC 15	SFC 15	// Write Consistent Data to a Standard DP Slave
"DIS_AIRT"	SFC 41	SFC 41	// Delay the Higher Priority Interrupts and Asynchronous Errors
"EN_AIRT"	SFC 42	SFC 42	// Enable Higher Priority Interrupts and Asynchronous Errors
"LGC_GADR"	SFC 49	SFC 49	// Query the Module Slot Belonging to a Logical Address
"RDSYSST"	SFC 51	SFC 51	// Read a System Status List or Partial List
"WR_REC"	SFC 58	SFC 58	// Write Data Record
"RD_REC"	SFC 59	SFC 59	// Read a Data Record
"T1"	T 1	TIMER
"T2"	T 2	TIMER
"T3"	T 3	TIMER
"T4"	T 4	TIMER
"T5"	T 5	TIMER
"T6"	T 6	TIMER
"T7"	T 7	TIMER
"T8"	T 8	TIMER
"T9"	T 9	TIMER
"T10"	T 10	TIMER
"Linea 1 Vuota"	T 22	TIMER
"Linea 2 Vuota"	T 23	TIMER
"T100"	T 100	TIMER
"T101"	T 101	TIMER
"T102"	T 102	TIMER
"T103"	T 103	TIMER
"T104"	T 104	TIMER
"T105"	T 105	TIMER
"T106"	T 106	TIMER
"T107"	T 107	TIMER
"T108"	T 108	TIMER
"T109"	T 109	TIMER
"T110"	T 110	TIMER
"T111"	T 111	TIMER
"T112"	T 112	TIMER
"T113"	T 113	TIMER
"T114"	T 114	TIMER
"T115"	T 115	TIMER
"T116"	T 116	TIMER
"T117"	T 117	TIMER
"T120"	T 120	TIMER
"T121"	T 121	TIMER
"T122"	T 122	TIMER
"T123"	T 123	TIMER
"T124"	T 124	TIMER
"T125"	T 125	TIMER	// TEMPO CHIUSURA ALLINEATORE LINEA 1
"MM4_Control_Word"	UDT 1	UDT 1
"MM4_Status_Word"	UDT 2	UDT 2
"UDT_Manuali"	UDT 100	UDT 100
"UDT_Allarmi"	UDT 101	UDT 101
"UDT_Segnalazioni"	UDT 102	UDT 102
"UDT_PARAM_INV"	UDT 200	UDT 200
"UDT_PKW_INV"	UDT 201	UDT 201
"UDT_Inverter_Record"	UDT 202	UDT 202
"UDT_String64"	UDT 271	UDT 271
"UDT_ANY_Pointer"	UDT 274	UDT 274
"VAT_1"	VAT 1	
"TestEthernet"	VAT 2	
"VAT_Code"	VAT 3	
"VAT_Dati"	VAT 4	
END_SYMBOL_TABLE

TYPE "MM4_Control_Word"	// UDT 1
AUTHOR : PROTEKNO
FAMILY : Profibus
NAME : MM4
VERSION : 0.1
  STRUCT
   Bit_8 : BOOL ;	//1=Jog right on/ 0=Jog right off
   Bit_9 : BOOL ;	//1=Jog left on / 0=Jog left off
   Bit_10 : BOOL ;	//1=Setpoint valid / 0=Setpoint invalid
   Bit_11 : BOOL ;	//1=Setpoint inverted/ 0=Setpoint is not inverted
   Bit_12 : BOOL ;	//-
   Bit_13 : BOOL ;	//1=Motor potentiometer UP / 0=No meaning
   Bit_14 : BOOL ;	//1=Motor potentiometer Down / 0=No meaning
   Bit_15 : BOOL ;	//1=Local control active(BOP/AOP) / 0=Remote control active
   Bit_0 : BOOL ;	//1=On/ 0=OFF
   Bit_1 : BOOL ;	//1=Operating condition/ 0=OFF2 - pulse disable
   Bit_2 : BOOL ;	//1=Operating condition/ 0=OFF3 - Rapid stop
   Bit_3 : BOOL ;	//1=Enable operation/ 0=Disable operation
   Bit_4 : BOOL ;	//1=Operating condition/ 0=Disable RFG
   Bit_5 : BOOL ;	//1=Enable RFG / 0=Stop RFG
   Bit_6 : BOOL ;	//1=Enable setpoint/ 0=Disable setpoint
   Bit_7 : BOOL ;	//1=fault acknowledge / 0=No meaning
  END_STRUCT ;	
END_TYPE

TYPE "MM4_Status_Word"	// UDT 2
AUTHOR : PROTEKNO
FAMILY : Profibus
NAME : MM4
VERSION : 0.1
  STRUCT
   Bit_8 : BOOL ;	//1=No setpoint-act.val. deviation/ 0=setpoint-act.val. deviation
   Bit_9 : BOOL ;	//1=Master control requested/ 0=Local operation
   Bit_10 : BOOL ;	//1=fmax reached/ 0=fmax not reached
   Bit_11 : BOOL ;	//1= / 0=Alarm:Motor at current limit
   Bit_12 : BOOL ;	//1= / 0=Motor holding brake
   Bit_13 : BOOL ;	//1= / 0=Motor overload
   Bit_14 : BOOL ;	//1= CW rotation / 0= CCW rotation
   Bit_15 : BOOL ;	//1= /0=Converter overload
   Bit_0 : BOOL ;	//1=Ready for On/ 0=Not ready for On
   Bit_1 : BOOL ;	//1=Ready for run/  0=Not ready for run
   Bit_2 : BOOL ;	//1=Operation enabled/ 0=Operation disabled
   Bit_3 : BOOL ;	//1=Fault active / 0=No fault active
   Bit_4 : BOOL ;	//1=No OFF2 command applied / 0=OFF2 command applied
   Bit_5 : BOOL ;	//1=No OFF3 command applied / 0=OFF3 command applied
   Bit_6 : BOOL ;	//1=Starting lockout / 0=No Starting lockout
   Bit_7 : BOOL ;	//1=Alarm is active / 0= Alarm is active
  END_STRUCT ;	
END_TYPE

TYPE "UDT_Manuali"	// UDT 100
VERSION : 0.0
  STRUCT
   Man001 : BOOL ;	// Comando Motore M1 estrattore EIDOS
   Man002 : BOOL ;	// Comando Motore M2 estrattore EIDOS
   Man003 : BOOL ;
   Man004 : BOOL ;
   Man005 : BOOL ;	// Comando salita traslatore
   Man006 : BOOL ;	// Comando discesa traslatore
   Man007 : BOOL ;	// Comando Motore M3 catena traslatore
   Man008 : BOOL ;
   Man009 : BOOL ;
   Man010 : BOOL ;	// Comando motore M20 rulliera 4 trofili
   Man011 : BOOL ;	// Comando motore M21 rulliera 4 trofili
   Man012 : BOOL ;	// Comando motore M22 rulliera 4 trofili
   Man013 : BOOL ;	// Comando motore M23 rulliera 4 trofili
   Man014 : BOOL ;	// Comando motore M24 rulliera 4 trofili
   Man015 : BOOL ;	// Comando motore M25 rulliera 4 trofili
   Man016 : BOOL ;
   Man017 : BOOL ;
   Man018 : BOOL ;
   Man019 : BOOL ;
   Man020 : BOOL ;	//Comando salita nastro prelievo Linea 1
   Man021 : BOOL ;	//Comando discesa nastro prelievo Linea 1
   Man022 : BOOL ;	//Comando motore M11 catena basculante prelievo cadenzatore Linea 1
   Man023 : BOOL ;	//Comando motore M10 catena cadenzatore linea 1
   Man024 : BOOL ;	//Comando motore M9  catena basculante deposito cadenzatore Linea 1
   Man025 : BOOL ;	//Comando motore M8  cadenzatore Linea 1
   Man026 : BOOL ;	//Comando salita nastro deposito Linea 1
   Man027 : BOOL ;	//Comando discesa nastro deposito Linea 1
   Man028 : BOOL ;
   Man029 : BOOL ;
   Man030 : BOOL ;	//Comando motore M27 rulliera 1 ingresso estrusore Linea 1
   Man031 : BOOL ;	//Comando motore M28 rulliera 2 ingresso estrusore Linea 1
   Man032 : BOOL ;	//Comando motore M29 rulliera 3 ingresso estrusore Linea 1
   Man033 : BOOL ;	//Comando chiusura allinetore M27
   Man034 : BOOL ;	//Comando motore M32 rulliera 1 uscita estrusore Linea 1
   Man035 : BOOL ;	//Comando motore M33 rulliera 2 uscita estrusore Linea 1
   Man036 : BOOL ;	//Comando motore M34 rulliera 3 uscita estrusore Linea 1
   Man037 : BOOL ;	//Comando motore M35 rulliera 4 uscita estrusore Linea 1
   Man038 : BOOL ;
   Man039 : BOOL ;
   Man040 : BOOL ;	//Comando salita nastro prelievo scarico A Linea 1
   Man041 : BOOL ;	//Comando discesa nastro prelievo scarico A Linea 1
   Man042 : BOOL ;	//Comando motore M12 catena 1 scarico A linea 1
   Man043 : BOOL ;	//Comando motore M13 catena 2 scarico A linea 1
   Man044 : BOOL ;
   Man045 : BOOL ;	//Comando salita nastro prelievo scarico B Linea 1
   Man046 : BOOL ;	//Comando discesa nastro prelievo scarico B Linea 1
   Man047 : BOOL ;	//Comando motore M14 catena 1 scarico B linea 1
   Man048 : BOOL ;	//Comando motore M15 catena 2 scarico B linea 1
   Man049 : BOOL ;
   Man050 : BOOL ;	//Comando salita nastro prelievo Linea 2
   Man051 : BOOL ;	//Comando discesa nastro prelievo Linea 2
   Man052 : BOOL ;	//Comando motore M4 catena basculante prelievo cadenzatore Linea 2
   Man053 : BOOL ;	//Comando motore M5 catena cadenzatore linea 2
   Man054 : BOOL ;	//Comando motore M6  catena basculante deposito cadenzatore Linea 2
   Man055 : BOOL ;	//Comando motore M7  cadenzatore Linea 2
   Man056 : BOOL ;	//Comando salita nastro deposito Linea 2
   Man057 : BOOL ;	//Comando discesa nastro deposito Linea 2
   Man058 : BOOL ;
   Man059 : BOOL ;
   Man060 : BOOL ;	//Comando motore M25 rulliera 1 ingresso estrusore Linea 2
   Man061 : BOOL ;	//Comando motore M26 rulliera 2 ingresso estrusore Linea 2
   Man062 : BOOL ;
   Man063 : BOOL ;
   Man064 : BOOL ;
   Man065 : BOOL ;	//Comando motore M30 rulliera 1 uscita estrusore Linea 2
   Man066 : BOOL ;	//Comando motore M31 rulliera 2 uscita estrusore Linea 2
   Man067 : BOOL ;	//Comando motore M16 cadenzatore scarico A Linea 2
   Man068 : BOOL ;	//Comando motore M17 catena scarico A linea 2
   Man069 : BOOL ;	//Comando motore M18 cadenzatore scarico B Linea 2
   Man070 : BOOL ;	//Comando motore M19 catena scarico B linea 2
   Man071 : BOOL ;
   Man072 : BOOL ;
   Man073 : BOOL ;
   Man074 : BOOL ;
   Man075 : BOOL ;
   Man076 : BOOL ;
   Man077 : BOOL ;
   Man078 : BOOL ;
   Man079 : BOOL ;
   Man080 : BOOL ;
   Man081 : BOOL ;
   Man082 : BOOL ;
   Man083 : BOOL ;
   Man084 : BOOL ;
   Man085 : BOOL ;
   Man086 : BOOL ;
   Man087 : BOOL ;
   Man088 : BOOL ;
   Man089 : BOOL ;
   Man090 : BOOL ;
   Man091 : BOOL ;
   Man092 : BOOL ;
   Man093 : BOOL ;
   Man094 : BOOL ;
   Man095 : BOOL ;
   Man096 : BOOL ;
   Man097 : BOOL ;
   Man098 : BOOL ;
   Man099 : BOOL ;
   Man100 : BOOL ;
   Man101 : BOOL ;
   Man102 : BOOL ;
   Man103 : BOOL ;
   Man104 : BOOL ;
   Man105 : BOOL ;
   Man106 : BOOL ;
   Man107 : BOOL ;
   Man108 : BOOL ;
   Man109 : BOOL ;
   Man110 : BOOL ;
   Man111 : BOOL ;
   Man112 : BOOL ;
   Man113 : BOOL ;
   Man114 : BOOL ;
   Man115 : BOOL ;
   Man116 : BOOL ;
   Man117 : BOOL ;
   Man118 : BOOL ;
   Man119 : BOOL ;
   Man120 : BOOL ;
   Man121 : BOOL ;
   Man122 : BOOL ;
   Man123 : BOOL ;
   Man124 : BOOL ;
   Man125 : BOOL ;
   Man126 : BOOL ;
   Man127 : BOOL ;
   Man128 : BOOL ;
  END_STRUCT ;	
END_TYPE

TYPE "UDT_Allarmi"	// UDT 101
VERSION : 0.0
  STRUCT 	// UDT definizione allarmi
   Msg_001 : BOOL ;	//INTERVENTO TERMICO "KMC1" (E0.0)
   Msg_002 : BOOL ;	//INTERVENTO TERMICO "KMC2" (E0.1)
   Msg_003 : BOOL ;	//INTERVENTO TERMICO "KMC3" (E0.2)
   Msg_004 : BOOL ;	//INTERVENTO TERMICO "KMC4" (E0.3)
   Msg_005 : BOOL ;	//INTERVENTO TERMICO "KMC5" (E0.4)
   Msg_006 : BOOL ;	//INTERVENTO TERMICO "KMC6" (E0.5)
   Msg_007 : BOOL ;	//INTERVENTO TERMICO "KMC7" (E0.6)
   Msg_008 : BOOL ;	//INTERVENTO TERMICO "KMC8" (E0.7)
   Msg_009 : BOOL ;	//INTERVENTO TERMICO "KMC9" (E1.0)
   Msg_010 : BOOL ;	//INTERVENTO TERMICO "KMC10" (E1.1)
   Msg_011 : BOOL ;	//INTERVENTO TERMICO "KMC11" (E1.2)
   Msg_012 : BOOL ;	//INTERVENTO TERMICO "KMC12" (E1.3)
   Msg_013 : BOOL ;	//INTERVENTO TERMICO "KMC13" (E1.4)
   Msg_014 : BOOL ;	//INTERVENTO TERMICO "KMC14" (E1.5)
   Msg_015 : BOOL ;	//INTERVENTO TERMICO "KMC15" (E1.6)
   Msg_016 : BOOL ;	//INTERVENTO TERMICO "KMC16" (E1.7)
   Msg_017 : BOOL ;	//INTERVENTO TERMICO "KMC17" (E2.0)
   Msg_018 : BOOL ;	//INTERVENTO TERMICO "KMC18" (E2.1)
   Msg_019 : BOOL ;	//INTERVENTO TERMICO "KMC19" (E2.2)
   Msg_020 : BOOL ;	//INTERVENTO TERMICO "KMC20" (E2.3)
   Msg_021 : BOOL ;	//INTERVENTO TERMICO "QF20" ALIM. INVERTER A1 "M20" (E3.0)
   Msg_022 : BOOL ;	//INTERVENTO TERMICO "QF21" ALIM. INVERTER A2 "M21" (E3.1)
   Msg_023 : BOOL ;	//INTERVENTO TERMICO "QF22" ALIM. INVERTER A3 "M22" (E3.2)
   Msg_024 : BOOL ;	//INTERVENTO TERMICO "QF23" ALIM. INVERTER A4 "M23" (E3.3)
   Msg_025 : BOOL ;	//INTERVENTO TERMICO "QF24" ALIM. INVERTER A5 "M24" (E3.4)
   Msg_026 : BOOL ;	//INTERVENTO TERMICO "QF25" ALIM. INVERTER A6 "M25" (E3.5)
   Msg_027 : BOOL ;	//INTERVENTO TERMICO "QF26" ALIM. INVERTER A7 "M26" (E3.6)
   Msg_028 : BOOL ;	//INTERVENTO TERMICO "QF27" ALIM. INVERTER A8 "M27" (E3.7)
   Msg_029 : BOOL ;	//INTERVENTO TERMICO "QF28" ALIM. INVERTER A9 "M28" (E4.0)
   Msg_030 : BOOL ;	//INTERVENTO TERMICO "QF29" ALIM. INVERTER A10 "M29" (E4.1)
   Msg_031 : BOOL ;	//INTERVENTO TERMICO "QF30" ALIM. INVERTER A11 "M30" (E4.2)
   Msg_032 : BOOL ;	//INTERVENTO TERMICO "QF31" ALIM. INVERTER A12 "M31" (E4.3)
   Msg_033 : BOOL ;	//INTERVENTO TERMICO "QF32" ALIM. INVERTER A13 "M32" (E4.4)
   Msg_034 : BOOL ;	//INTERVENTO TERMICO "QF33" ALIM. INVERTER A14 "M33" (E4.5)
   Msg_035 : BOOL ;	//INTERVENTO TERMICO "QF34" ALIM. INVERTER A15 "M34" (E4.6)
   Msg_036 : BOOL ;	//INTERVENTO TERMICO "QF35" ALIM. INVERTER A16 "M35" (E4.7)
   Msg_037 : BOOL ;	//INTERVENTO TERMICO "QF36"(E5.0)
   Msg_038 : BOOL ;
   Msg_039 : BOOL ;
   Msg_040 : BOOL ;
   Msg_041 : BOOL ;	//INTERVENTO PROTEZIONE "QF6" VENTILAZIONE QUADRO (E5.1)
   Msg_042 : BOOL ;	//INTERVENTO PROTEZIONE "QF8"  (E5.2)
   Msg_043 : BOOL ;	//INTERVENTO PROTEZIONE "QF19" ALIM. CIRCUITI D'EMERGENZA  (E5.3)
   Msg_044 : BOOL ;	//INTERVENTO PROTEZIONE "QF10" ALIM. COMANDI QUADRO (E5.4)
   Msg_045 : BOOL ;	//INTERVENTO PROTEZIONE "QF11" ALIM. COMANDI JP1  (E5.5)
   Msg_046 : BOOL ;	//INTERVENTO PROTEZIONE "QF12" ALIM. COMANDI JP2  (E5.6)
   Msg_047 : BOOL ;	//INTERVENTO PROTEZIONE "QF13" ALIM. COMANDI JP3  (E5.7)
   Msg_048 : BOOL ;
   Msg_049 : BOOL ;	//FAULT NODO PROFIBUS 3 (INVERTER "M20")
   Msg_050 : BOOL ;	//FAULT NODO PROFIBUS 4 (INVERTER "M21")
   Msg_051 : BOOL ;	//FAULT NODO PROFIBUS 5 (INVERTER "M22")
   Msg_052 : BOOL ;	//FAULT NODO PROFIBUS 6 (INVERTER "M23")
   Msg_053 : BOOL ;	//FAULT NODO PROFIBUS 7 (INVERTER "M24")
   Msg_054 : BOOL ;	//FAULT NODO PROFIBUS 8 (INVERTER "M25")
   Msg_055 : BOOL ;	//FAULT NODO PROFIBUS 9 (INVERTER "M26")
   Msg_056 : BOOL ;	//FAULT NODO PROFIBUS 10 (INVERTER "M27")
   Msg_057 : BOOL ;	//FAULT NODO PROFIBUS 11 (INVERTER "M28")
   Msg_058 : BOOL ;	//FAULT NODO PROFIBUS 12 (INVERTER "M29")
   Msg_059 : BOOL ;	//FAULT NODO PROFIBUS 13 (INVERTER "M30")
   Msg_060 : BOOL ;	//FAULT NODO PROFIBUS 14 (INVERTER "M31")
   Msg_061 : BOOL ;	//FAULT NODO PROFIBUS 15 (INVERTER "M32")
   Msg_062 : BOOL ;	//FAULT NODO PROFIBUS 16 (INVERTER "M33")
   Msg_063 : BOOL ;	//FAULT NODO PROFIBUS 17 (INVERTER "M34")
   Msg_064 : BOOL ;	//FAULT NODO PROFIBUS 18 (INVERTER "M35")
   Msg_065 : BOOL ;	//FAULT NODO PROFIBUS 24 (DP/DP COUPLER FORNO)
   Msg_066 : BOOL ;	//FAULT NODO PROFIBUS 25 (ET200S - BOX JP1)
   Msg_067 : BOOL ;	//FAULT NODO PROFIBUS 26 (ET200S - BOX JP2)
   Msg_068 : BOOL ;	//FAULT NODO PROFIBUS 27 (ET200S - BOX JP3)
   Msg_069 : BOOL ;
   Msg_070 : BOOL ;	//TIMEOUT FINECORSA ALTO TRASLATORE 4 PEZZI (E20.0, E20.2)
   Msg_071 : BOOL ;	//TIMEOUT FINECORSA BASSO TRASLATORE 4 PEZZI (E20.1, E20.3)
   Msg_072 : BOOL ;	//TIMEOUT FINECORSA ALTO CATENE INGRESSO 4 PEZZI LINEA 2 (E21.4, E21.6)
   Msg_073 : BOOL ;	//TIMEOUT FINECORSA BASSO CATENE INGRESSO 4 PEZZI LINEA 2 (E21.5, E21.7)
   Msg_074 : BOOL ;	//TIMEOUT FINECORSA ALTO CATENE USCITA CADENZATORE LINEA 2 (E21.0, E21.2)
   Msg_075 : BOOL ;	//TIMEOUT FINECORSA BASSO CATENE USCITA CADENZATORE LINEA 2 (E21.1, E21.3)
   Msg_076 : BOOL ;	//TIMEOUT FINECORSA ALTO CATENE INGRESSO 4 PEZZI LINEA 1 (E22.0, E22.2)
   Msg_077 : BOOL ;	//TIMEOUT FINECORSA BASSO CATENE INGRESSO 4 PEZZI LINEA 1 (E22.1, E22.3)
   Msg_078 : BOOL ;	//TIMEOUT FINECORSA ALTO CATENE USCITA CADENZATORE LINEA 1 (E22.4, E22.6)
   Msg_079 : BOOL ;	//TIMEOUT FINECORSA BASSO CATENE USCITA CADENZATORE LINEA 1 (E22.5, E22.7)
   Msg_080 : BOOL ;	//TIMEOUT FINECORSA ALTO CATENE ACCUMULO "A" LINEA 1 (E25.0, E25.2)
   Msg_081 : BOOL ;	//TIMEOUT FINECORSA BASSO CATENE ACCUMULO "A" LINEA 1 (E25.1, E25.3)
   Msg_082 : BOOL ;	//TIMEOUT FINECORSA ALTO CATENE ACCUMULO "B" LINEA 1 (E25.4, E25.6)
   Msg_083 : BOOL ;	//TIMEOUT FINECORSA BASSO CATENE ACCUMULO "B" LINEA 1 (E25.5, E25.7)
   Msg_084 : BOOL ;	//TIMEOUT SENSORE PASSO CADENZATORE INGRESSO LINEA 2 (E24.0)
   Msg_085 : BOOL ;	//TIMEOUT SENSORE PASSO CADENZATORE INGRESSO LINEA 1 (E24.1)
   Msg_086 : BOOL ;	//TIMEOUT SENSORE PASSO CADENZATORE ACCUMULO "A" LINEA 2 (E27.2)
   Msg_087 : BOOL ;	//TIMEOUT SENSORE PASSO CADENZATORE ACCUMULO "B" LINEA 2 (E27.3)
   Msg_088 : BOOL ;
   Msg_089 : BOOL ;	//CADENZATORE INGRESSO LINEA 2 NON IN FASE (E24.0)
   Msg_090 : BOOL ;	//CADENZATORE INGRESSO LINEA 1 NON IN FASE (E24.1)
   Msg_091 : BOOL ;	//CADENZATORE ACCUMULO "A" LINEA 2 NON IN FASE (E27.2)
   Msg_092 : BOOL ;	//CADENZATORE ACCUMULO "B" LINEA 2 NON IN FASE (E27.3)
   Msg_093 : BOOL ;	//FOTOCELLULA ARRESTO PACCO 4 FILE TRASLATORE E' RIMASTA IMPEGNATA (E20.4)
   Msg_094 : BOOL ;	//FOTOCELLULA ARRESTO PACCO 4 FILE DAVANTI LINEA 2 E' RIMASTA IMPEGNATA (E23.6)
   Msg_095 : BOOL ;	//FOTOCELLULA ARRESTO PACCO 4 FILE DAVANTI LINEA 1 E' RIMASTA IMPEGNATA (E23.7)
   Msg_096 : BOOL ;	//FOTOCELLULA ARRESTO BARRA DAVANTI CADENZATORE LINEA 2 E' RIMASTA IMPEGNATA (E23
   Msg_097 : BOOL ;	//FOTOCELLULA ARRESTO BARRA DAVANTI CADENZATORE LINEA 1 E' RIMASTA IMPEGNATA (E23
   Msg_098 : BOOL ;	//FOTOCELLULA ARRESTO BARRA SU RULLIERA 1 INGRESSO ESTR. LINEA 2 E' RIMASTA IMPEG
   Msg_099 : BOOL ;	//FOTOCELLULA ARRESTO BARRA SU RULLIERA 1 INGRESSO ESTR. LINEA 1 E' RIMASTA IMPEG
   Msg_100 : BOOL ;	//FOTOCELLULA ARRESTO BARRA SU CADENZATORE ACCUMULO "A" LINEA 2 E' RIMASTA IMPEGN
   Msg_101 : BOOL ;	//FOTOCELLULA ARRESTO BARRA SU CADENZATORE ACCUMULO "B" LINEA 2 E' RIMASTA IMPEGN
   Msg_102 : BOOL ;	//FOTOCELLULA ARRESTO BARRA SU DEVIATORE ACCUMULO "A" LINEA 1 E' RIMASTA IMPEGNAT
   Msg_103 : BOOL ;	//FOTOCELLULA ARRESTO BARRA SU DEVIATORE ACCUMULO "B" LINEA 1 E' RIMASTA IMPEGNAT
   Msg_104 : BOOL ;
   Msg_105 : BOOL ;	//TIMEOUT CICLO TRASFERITORE O MANCATA LETTURA FOTOCELLULA ARRESTO CATENE (E20.4)
   Msg_106 : BOOL ;	//TIMEOUT CICLO TRASFERIMENTO 4 BARRE VERSO LINEA 2 O MANCATA LETTURA FOTOCELLULA
   Msg_107 : BOOL ;	//TIMEOUT CICLO TRASFERIMENTO 4 BARRE VERSO LINEA 1 O MANCATA LETTURA FOTOCELLULA
   Msg_108 : BOOL ;	//TIMEOUT CICLO ALIMENTAZIONE CADENZATORE LINEA 2 O MANCATA LETTURA FOTOCELLULA (
   Msg_109 : BOOL ;	//TIMEOUT CICLO ALIMENTAZIONE CADENZATORE LINEA 1 O MANCATA LETTURA FOTOCELLULA (
   Msg_110 : BOOL ;	//LINEA ACCUMULO "A" INFERIORE PIENA
   Msg_111 : BOOL ;	//LINEA ACCUMULO "A" SUPERIORE PIENA
   Msg_112 : BOOL ;	//LINEA ACCUMULO "B" INFERIORE PIENA
   Msg_113 : BOOL ;	//LINEA ACCUMULO "B" SUPERIORE PIENA
   Msg_114 : BOOL ;	//INVERTER A1 MOTORE "M20" IN ALLARME
   Msg_115 : BOOL ;	//INVERTER A2 MOTORE "M21" IN ALLARME
   Msg_116 : BOOL ;	//INVERTER A3 MOTORE "M22" IN ALLARME
   Msg_117 : BOOL ;	//INVERTER A4 MOTORE "M23" IN ALLARME
   Msg_118 : BOOL ;	//INVERTER A5 MOTORE "M24" IN ALLARME
   Msg_119 : BOOL ;	//INVERTER A6 MOTORE "M25" IN ALLARME
   Msg_120 : BOOL ;	//INVERTER A7 MOTORE "M26" IN ALLARME
   Msg_121 : BOOL ;	//INVERTER A8 MOTORE "M27" IN ALLARME
   Msg_122 : BOOL ;	//INVERTER A9 MOTORE "M28" IN ALLARME
   Msg_123 : BOOL ;	//INVERTER A10 MOTORE "M29" IN ALLARME
   Msg_124 : BOOL ;	//INVERTER A11 MOTORE "M30" IN ALLARME
   Msg_125 : BOOL ;	//INVERTER A12 MOTORE "M31" IN ALLARME
   Msg_126 : BOOL ;	//INVERTER A13 MOTORE "M32" IN ALLARME
   Msg_127 : BOOL ;	//INVERTER A14 MOTORE "M33" IN ALLARME
   Msg_128 : BOOL ;	//INVERTER A15 MOTORE "M34" IN ALLARME
   Msg_129 : BOOL ;	//INVERTER A16 MOTORE "M35" IN ALLARME
   Msg_130 : BOOL ;
   Msg_131 : BOOL ;
   Msg_132 : BOOL ;
   Msg_133 : BOOL ;
   Msg_134 : BOOL ;
   Msg_135 : BOOL ;
   Msg_136 : BOOL ;
   Msg_137 : BOOL ;
   Msg_138 : BOOL ;
   Msg_139 : BOOL ;
   Msg_140 : BOOL ;
   Msg_141 : BOOL ;
   Msg_142 : BOOL ;
   Msg_143 : BOOL ;
   Msg_144 : BOOL ;
   Msg_145 : BOOL ;
   Msg_146 : BOOL ;
   Msg_147 : BOOL ;
   Msg_148 : BOOL ;
   Msg_149 : BOOL ;
   Msg_150 : BOOL ;
   Msg_151 : BOOL ;
   Msg_152 : BOOL ;
   Msg_153 : BOOL ;
   Msg_154 : BOOL ;
   Msg_155 : BOOL ;
   Msg_156 : BOOL ;
   Msg_157 : BOOL ;
   Msg_158 : BOOL ;
   Msg_159 : BOOL ;
   Msf_160 : BOOL ;
  END_STRUCT ;	
END_TYPE

TYPE "UDT_Segnalazioni"	// UDT 102
VERSION : 0.0
  STRUCT 	// Descrizione del tipo
   Msg_1001 : BOOL ;
   Msg_1002 : BOOL ;
   Msg_1003 : BOOL ;
   Msg_1004 : BOOL ;
   Msg_1005 : BOOL ;
   Msg_1006 : BOOL ;
   Msg_1007 : BOOL ;
   Msg_1008 : BOOL ;
   Msg_1009 : BOOL ;
   Msg_1010 : BOOL ;
   Msg_1011 : BOOL ;
   Msg_1012 : BOOL ;
   Msg_1013 : BOOL ;
   Msg_1014 : BOOL ;
   Msg_1015 : BOOL ;
   Msg_1016 : BOOL ;
   Msg_1017 : BOOL ;
   Msg_1018 : BOOL ;
   Msg_1019 : BOOL ;
   Msg_1020 : BOOL ;
   Msg_1021 : BOOL ;
   Msg_1022 : BOOL ;
   Msg_1023 : BOOL ;
   Msg_1024 : BOOL ;
   Msg_1025 : BOOL ;
   Msg_1026 : BOOL ;
   Msg_1027 : BOOL ;
   Msg_1028 : BOOL ;
   Msg_1029 : BOOL ;
   Msg_1030 : BOOL ;
   Msg_1031 : BOOL ;
   Msg_1032 : BOOL ;
   Msg_1033 : BOOL ;
   Msg_1034 : BOOL ;
   Msg_1035 : BOOL ;
   Msg_1036 : BOOL ;
   Msg_1037 : BOOL ;
   Msg_1038 : BOOL ;
   Msg_1039 : BOOL ;
   Msg_1040 : BOOL ;
   Msg_1041 : BOOL ;
   Msg_1042 : BOOL ;
   Msg_1043 : BOOL ;
   Msg_1044 : BOOL ;
   Msg_1045 : BOOL ;
   Msg_1046 : BOOL ;
   Msg_1047 : BOOL ;
   Msg_1048 : BOOL ;
   Msg_1049 : BOOL ;
   Msg_1050 : BOOL ;
   Msg_1051 : BOOL ;
   Msg_1052 : BOOL ;
   Msg_1053 : BOOL ;
   Msg_1054 : BOOL ;
   Msg_1055 : BOOL ;
   Msg_1056 : BOOL ;
   Msg_1057 : BOOL ;
   Msg_1058 : BOOL ;
   Msg_1059 : BOOL ;
   Msg_1060 : BOOL ;
   Msg_1061 : BOOL ;
   Msg_1062 : BOOL ;
   Msg_1063 : BOOL ;
   Msg_1064 : BOOL ;
   Msg_1065 : BOOL ;
   Msg_1066 : BOOL ;
   Msg_1067 : BOOL ;
   Msg_1068 : BOOL ;
   Msg_1069 : BOOL ;
   Msg_1070 : BOOL ;
   Msg_1071 : BOOL ;
   Msg_1072 : BOOL ;
   Msg_1073 : BOOL ;
   Msg_1074 : BOOL ;
   Msg_1075 : BOOL ;
   Msg_1076 : BOOL ;
   Msg_1077 : BOOL ;
   Msg_1078 : BOOL ;
   Msg_1079 : BOOL ;
   Msg_1080 : BOOL ;
   Msg_1081 : BOOL ;
   Msg_1082 : BOOL ;
   Msg_1083 : BOOL ;
   Msg_1084 : BOOL ;
   Msg_1085 : BOOL ;
   Msg_1086 : BOOL ;
   Msg_1087 : BOOL ;
   Msg_1088 : BOOL ;
   Msg_1089 : BOOL ;
   Msg_1090 : BOOL ;
   Msg_1091 : BOOL ;
   Msg_1092 : BOOL ;
   Msg_1093 : BOOL ;
   Msg_1094 : BOOL ;
   Msg_1095 : BOOL ;
   Msg_1096 : BOOL ;
   Msg_1097 : BOOL ;
   Msg_1098 : BOOL ;
   Msg_1099 : BOOL ;
   Msg_1100 : BOOL ;
   Msg_1101 : BOOL ;
   Msg_1102 : BOOL ;
   Msg_1103 : BOOL ;
   Msg_1104 : BOOL ;
   Msg_1105 : BOOL ;
   Msg_1106 : BOOL ;
   Msg_1107 : BOOL ;
   Msg_1108 : BOOL ;
   Msg_1109 : BOOL ;
   Msg_1110 : BOOL ;
   Msg_1111 : BOOL ;
   Msg_1112 : BOOL ;
   Msg_1113 : BOOL ;
   Msg_1114 : BOOL ;
   Msg_1115 : BOOL ;
   Msg_1116 : BOOL ;
   Msg_1117 : BOOL ;
   Msg_1118 : BOOL ;
   Msg_1119 : BOOL ;
   Msg_1120 : BOOL ;
   Msg_1121 : BOOL ;
   Msg_1122 : BOOL ;
   Msg_1123 : BOOL ;
   Msg_1124 : BOOL ;
   Msg_1125 : BOOL ;
   Msg_1126 : BOOL ;
   Msg_1127 : BOOL ;
   Msg_1128 : BOOL ;
   Msg_1129 : BOOL ;
   Msg_1130 : BOOL ;
   Msg_1131 : BOOL ;
   Msg_1132 : BOOL ;
   Msg_1133 : BOOL ;
   Msg_1134 : BOOL ;
   Msg_1135 : BOOL ;
   Msg_1136 : BOOL ;
   Msg_1137 : BOOL ;
   Msg_1138 : BOOL ;
   Msg_1139 : BOOL ;
   Msg_1140 : BOOL ;
   Msg_1141 : BOOL ;
   Msg_1142 : BOOL ;
   Msg_1143 : BOOL ;
   Msg_1144 : BOOL ;
   Msg_1145 : BOOL ;
   Msg_1146 : BOOL ;
   Msg_1147 : BOOL ;
   Msg_1148 : BOOL ;
   Msg_1149 : BOOL ;
   Msg_1150 : BOOL ;
   Msg_1151 : BOOL ;
   Msg_1152 : BOOL ;
   Msg_1153 : BOOL ;
   Msg_1154 : BOOL ;
   Msg_1155 : BOOL ;
   Msg_1156 : BOOL ;
   Msg_1157 : BOOL ;
   Msg_1158 : BOOL ;
   Msg_1159 : BOOL ;
   Msg_1160 : BOOL ;
  END_STRUCT ;	
END_TYPE

TYPE "UDT_PARAM_INV"	// UDT 200
VERSION : 0.0
  STRUCT
   Job : BYTE ;	//Job richiesto 0 niente 2 lettura dword 3 scrittura dword
   NumParam : INT ;	//Numero paramentro
   NumInd : INT ;	//Indice
   Val : REAL ;	//Valore da scrivere
   JobStatus : WORD ;	//Esisto
   RetVal : REAL ;	//Valore letto dal parametro
  END_STRUCT ;	
END_TYPE

TYPE "UDT_PKW_INV"	// UDT 201
AUTHOR : Filip1
FAMILY : INVERTER
NAME : PKW
VERSION : 0.0
  STRUCT
   PKE : WORD ;	//Parameter ID
   IND : WORD ;	//Index
   PWE : DWORD ;	//Parameter value
  END_STRUCT ;	
END_TYPE

TYPE "UDT_Inverter_Record"	// UDT 202
VERSION : 0.0
  STRUCT
   SetpointFreq : REAL ;	//r20
   ActualFreq : REAL ;	//r21
   RmpSpeed : REAL ;	//r22
   OutFreq : REAL ;	//r24
   OutVoltage : REAL ;	//r25
   DCBusVoltage : REAL ;	//r26
   OutCurrent : REAL ;	//r27
   Coppia : REAL ;	//r31    no su MM420
   Potenza : REAL ;	//r32    no su MM420
   MotorTemp : REAL ;	//r35    no su MM420
   InverterTemp : REAL ;	//r37
   EnergyCount : REAL ;	//r39
   ADC_1 : REAL ;	//r752.0
   ADC_2 : REAL ;	//r752.1 no su MM420
   CodAnomalia1 : INT ;	//r947.0
   CodAnomalia2 : INT ;	//r947.1
   CodAnomalia3 : INT ;	//r947.2
   CodAnomalia4 : INT ;	//r947.3
   CodErrore1 : INT ;	//r2110.0
   CodErrore2 : INT ;	//r2110.1
   CodErrore3 : INT ;	//r2110.2
   CodErrore4 : INT ;	//r2110.3
  END_STRUCT ;	
END_TYPE

TYPE "UDT_String64"	// UDT 271
VERSION : 0.0
  STRUCT
   DefLen : BYTE ;	//Lunghezza stringa dichiarata
   StrLen : BYTE ;	//Lunghezza stringa effettiva
   Str : ARRAY  [1 .. 64 ] OF CHAR ;	//Caratteri stringa
  END_STRUCT ;	
END_TYPE

TYPE "UDT_ANY_Pointer"	// UDT 274
VERSION : 0.0
  STRUCT
   ID_Any : BYTE  := B#16#10;	//ID tipo any
   DataType : BYTE ;
   Size : INT ;
   DB_Num : INT ;
   Address : DWORD ;
  END_STRUCT ;	
END_TYPE

// FB 125: know-how protected block, not included

FUNCTION_BLOCK "ReadParamInverters"	// FB 210
TITLE = Leggi parametri inverter
AUTHOR : Filip1
FAMILY : MM4
NAME : ReadInv
VERSION : 1.0
VAR_INPUT
  Addr : INT ;
END_VAR
VAR_IN_OUT
  RecParam : STRUCT
   SetpointFreq : REAL ;	//r20
   ActualFreq : REAL ;	//r21
   RmpSpeed : REAL ;	//r22
   OutFreq : REAL ;	//r24
   OutVoltage : REAL ;	//r25
   DCBusVoltage : REAL ;	//r26
   OutCurrent : REAL ;	//r27
   Coppia : REAL ;	//r31    no su MM420
   Potenza : REAL ;	//r32    no su MM420
   MotorTemp : REAL ;	//r35    no su MM420
   InverterTemp : REAL ;	//r37
   EnergyCount : REAL ;	//r39
   ADC_1 : REAL ;	//r752.0
   ADC_2 : REAL ;	//r752.1 no su MM420
   CodAnomalia1 : INT ;	//r947.0
   CodAnomalia2 : INT ;	//r947.1
   CodAnomalia3 : INT ;	//r947.2
   CodAnomalia4 : INT ;	//r947.3
   CodErrore1 : INT ;	//r2110.0
   CodErrore2 : INT ;	//r2110.1
   CodErrore3 : INT ;	//r2110.2
   CodErrore4 : INT ;	//r2110.3
  END_STRUCT ;
END_VAR
VAR
  ParamP : STRUCT
   Job : BYTE ;	//Job richiesto 0 niente 2 lettura dword 3 scrittura dword
   NumParam : INT ;	//Numero paramentro
   NumInd : INT ;	//Indice
   Val : REAL ;	//Valore da scrivere
   JobStatus : WORD ;	//Esisto
   RetVal : REAL ;	//Valore letto dal parametro
  END_STRUCT ;
  PKW_IN : ARRAY  [1 .. 4 ] OF WORD ;
  PKW_OUT : ARRAY  [1 .. 4 ] OF WORD ;
  Index : INT ;
  NumParamToRead : ARRAY  [1 .. 24 ] OF //Configurazione MM420
  INT  := 20, 21, 22, 24, 25, 26, 27, -1, -1, -1, 37, 39, 752, -1, 947, 947, 947, 947, 2110, 2110, 2110, 2110, 0, 0;	//Configurazione MM420
  IndParamToRead : ARRAY  [1 .. 24 ] OF INT  := 0, 0, 0, 0, 0, 0, 0, 0, 0, 0, 0, 0, 0, 1, 0, 1, 2, 3, 0, 1, 2, 3, 0, 0;
  ParamValue : ARRAY  [1 .. 24 ] OF DWORD ;
  Esito : BOOL ;
  ReadError : BOOL ;
END_VAR
VAR_TEMP
  Aux : WORD ;
  RetVal : DWORD ;
END_VAR
BEGIN
// body was compiled from an SCL source; compiled code not shown
END_FUNCTION_BLOCK

FUNCTION_BLOCK "FB_ReadParamLoop"	// FB 211
VERSION : 0.0
VAR
  ReadInvM20 : FB 210;
  ReadInvM21 : FB 210;
  ReadInvM22 : FB 210;
  ReadInvM23 : FB 210;
  ReadInvM24 : FB 210;
  ReadInvM25 : FB 210;
  ReadInvM26 : FB 210;
  ReadInvM27 : FB 210;
  ReadInvM28 : FB 210;
  ReadInvM29 : FB 210;
  ReadInvM30 : FB 210;
  ReadInvM31 : FB 210;
  ReadInvM32 : FB 210;
  ReadInvM33 : FB 210;
  ReadInvM34 : FB 210;
  ReadInvM35 : FB 210;
  Multiplex : INT ;
END_VAR
BEGIN
// body was compiled from an SCL source; compiled code not shown
END_FUNCTION_BLOCK

FUNCTION_BLOCK "FB_GestCodeEstrusori"	// FB 212
VERSION : 0.0
VAR_INPUT
  InserisciInCoda1 : BOOL ;	//Richiesta inserimento elemento in CODA 1
  EliminaDaCoda1 : BOOL ;	//Richiesta eliminazione elemento da CODA 1
  ValoreDaInsCoda1 : INT ;	//Valore da inserire in CODA 1
  InserisciInCoda2 : BOOL ;	//Richiesta inserimento elemento in CODA 2
  EliminaDaCoda2 : BOOL ;	//Richiesta eliminazione elemento da CODA 2
  ValoreDaInsCoda2 : INT ;	//Valore da inserire in CODA 2
END_VAR
VAR_OUTPUT
  PrimoInCoda1 : INT ;	//Elemento in cima alla CODA 1
  ContCoda1 : INT ;	//Numero elementi in CODA 1
  PrimoInCoda2 : INT ;	//Elemento in cima alla CODA 2
  ContCoda2 : INT ;	//Numero elementi in CODA 2
  Coda1Piena : BOOL ;	//Numero massimo di elementi in CODA1
  Coda1Vuota : BOOL ;	//Coda1 vuota
  Coda2Piena : BOOL ;	//Numero massimo di elementi in CODA2
  Coda2Vuota : BOOL ;	//Coda1 vuota
END_VAR
VAR
  Coda1 : ARRAY  [1 .. 16 ] OF //0: non presente; 1: Scarica su A; 2: Scarica su B
  INT ;	//0: non presente; 1: Scarica su A; 2: Scarica su B
  Coda2 : ARRAY  [1 .. 16 ] OF //0: non presente; 1: Scarica su A; 2: Scarica su B
  INT ;	//0: non presente; 1: Scarica su A; 2: Scarica su B
  AuxFronteIns1 : BOOL ;
  AuxFronteDel1 : BOOL ;
  AuxFronteIns2 : BOOL ;
  AuxFronteDel2 : BOOL ;
END_VAR
VAR_TEMP
  I : INT ;
END_VAR
BEGIN
// body was compiled from an SCL source; compiled code not shown
END_FUNCTION_BLOCK

FUNCTION_BLOCK "FB_LinkEthernet"	// FB 213
TITLE = Gestione ricezione stringa via ethernet di lunghezza variabile
//
//La funzione necessita di un collegamento TCP progettato.
//Il collegamento TCP deve essere configurato con le seguenti impostazioni:
//
//La funzione usa le seguenti funzioni di libreria:
//FC 5    AG_SEND v4.2    (funzione di libreria SIMATIC NET CP343)   
//FC 6    AG_RECV v4.7    (funzione di libreria SIMATIC NET CP343)
//
//UDT usate dalla funzione:
//UDT 271 UDT_String64  
//UDT 274 UDT_ANY_Pointer  
//
AUTHOR : Filip1
FAMILY : Ethernet
NAME : StrEth
VERSION : 1.0
VAR_INPUT
  ID : INT  := 1;	//ID del Collegamento ethernet TCP
  LAddr : WORD  := W#16#100;	//Address della CP343-1 ethernet TCP
  Cmd_SendStr : BOOL ;
  Cmd_EchoRcv : BOOL  := TRUE;	//Ritrasmette tutto quello che viene ricevuto
  SendStr : STRING  [64 ];
END_VAR
VAR_OUTPUT
  RcvStr : STRING  [64 ];
  RcvStrNew : BOOL ;	//E' stata ricevuta una nuova stringa (dura un ciclo)
  RcvL1Msg : BOOL ;	//La stringa ricevuta inizia per L1
  RcvL2Msg : BOOL ;	//La stringa ricevuta inizia per L2
  Ready : BOOL ;	//Connessione presente con il terminale e funz. pronta a ricevere
  Out_Error : BOOL ;	//Errore nelle connessione ethernt
END_VAR
VAR
  Send : STRUCT
   Start : BOOL ;
   Done : BOOL ;
   Error : BOOL ;
   Status : WORD ;
   LEN : INT ;
   Cont : INT ;
   ContErr : INT ;
   LastErr : WORD ;
  END_STRUCT ;
  Rcv : STRUCT
   Ndr : BOOL ;
   Error : BOOL ;
   Status : WORD ;
   LEN : INT ;
   Cont : INT ;
   ContErr : INT ;
   LastErr : WORD ;
   LenFcRx : INT ;
   Head : INT ;
   EthRxBuf : ARRAY  [1 .. 2 ] OF BYTE ;
  END_STRUCT ;
  RxWait : BOOL ;
  TxEchoRcv : BOOL ;
  SendStarted : BOOL ;
  TxOk : BOOL ;
  MemStrL1 : BOOL ;
  MemStrL2 : BOOL ;
  T_TimeoutRx : SFB 4;
  T_TimeoutTx : SFB 4;
  BufferTx : ARRAY  [1 .. 240 ] OF BYTE ;
  BufferRx : ARRAY  [1 .. 240 ] OF BYTE ;
END_VAR
VAR_TEMP
  P : ANY ;
  i : INT ;
  n : INT ;
END_VAR
BEGIN
// body was compiled from an SCL source; compiled code not shown
END_FUNCTION_BLOCK

FUNCTION "Allarmi" : VOID	// FC 1
NAME : Alarm
VERSION : 0.1
BEGIN
NETWORK
TITLE =
      A     "PULSANTE_RESET";
      FP    "M82.4";
      JNB   _001;
      CALL  "FC_ResetAllarmi" (
           Allarmi                  := "DB_OP".Allarmi);
_001: NOP   0;
NETWORK
TITLE = INTERVENTO TERMICO "KMC1" (E0.0)
      AN    "Termico_M1";
      S     "DB_OP".Allarmi.Msg_001;
NETWORK
TITLE = INTERVENTO TERMICO "KMC2" (E0.1)
      AN    "Termico_M2";
      S     "DB_OP".Allarmi.Msg_002;
NETWORK
TITLE = INTERVENTO TERMICO "KMC3" (E0.2)
      AN    "Termico_M3";
      S     "DB_OP".Allarmi.Msg_003;
NETWORK
TITLE = INTERVENTO TERMICO "KMC4" (E0.3)
      AN    "Termico_M4";
      S     "DB_OP".Allarmi.Msg_004;
NETWORK
TITLE = INTERVENTO TERMICO "KMC5" (E0.4)
      AN    "Termico_M5";
      S     "DB_OP".Allarmi.Msg_005;
NETWORK
TITLE = INTERVENTO TERMICO "KMC6" (E0.5)
      AN    "Termico_M6";
      S     "DB_OP".Allarmi.Msg_006;
NETWORK
TITLE = INTERVENTO TERMICO "KMC7" (E0.6)
      AN    "Termico_M7";
      S     "DB_OP".Allarmi.Msg_007;
NETWORK
TITLE = INTERVENTO TERMICO "KMC8" (E0.7)
      AN    "Termico_M8";
      S     "DB_OP".Allarmi.Msg_008;
NETWORK
TITLE = INTERVENTO TERMICO "KMC9" (E1.0)
      AN    "Termico_M9";
      S     "DB_OP".Allarmi.Msg_009;
NETWORK
TITLE = INTERVENTO TERMICO "KMC10" (E1.1)
      AN    "Termico_M10";
      S     "DB_OP".Allarmi.Msg_010;
NETWORK
TITLE = INTERVENTO TERMICO "KMC11" (E1.2)
      AN    "Termico_M11";
      S     "DB_OP".Allarmi.Msg_011;
NETWORK
TITLE = INTERVENTO TERMICO "KMC12" (E1.3)
      AN    "Termico_M12";
      S     "DB_OP".Allarmi.Msg_012;
NETWORK
TITLE = INTERVENTO TERMICO "KMC13" (E1.4)
      AN    "Termico_M13";
      S     "DB_OP".Allarmi.Msg_013;
NETWORK
TITLE = INTERVENTO TERMICO "KMC14" (E1.5)
      AN    "Termico_M14";
      S     "DB_OP".Allarmi.Msg_014;
NETWORK
TITLE = INTERVENTO TERMICO "KMC15" (E1.6)
      AN    "Termico_M15";
      S     "DB_OP".Allarmi.Msg_015;
NETWORK
TITLE = INTERVENTO TERMICO "KMC16" (E1.7)
      AN    "Termico_M16";
      S     "DB_OP".Allarmi.Msg_016;
NETWORK
TITLE = INTERVENTO TERMICO "KMC17" (E2.0)
      AN    "Termico_M17";
      S     "DB_OP".Allarmi.Msg_017;
NETWORK
TITLE = INTERVENTO TERMICO "KMC18" (E2.1)
      AN    "Termico_M18";
      S     "DB_OP".Allarmi.Msg_018;
NETWORK
TITLE = INTERVENTO TERMICO "KMC19" (E2.2)
      AN    "Termico_M19";
      S     "DB_OP".Allarmi.Msg_019;
NETWORK
TITLE = INTERVENTO TERMICO "KMC20" (E2.3)
      AN    "Termico_Avviatore_Spare";
      S     "DB_OP".Allarmi.Msg_020;
NETWORK
TITLE = INTERVENTO TERMICO "QF20" ALIM. INVERTER M20 (E3.0)
      AN    "QF20_Inverter_M20";
      S     "DB_OP".Allarmi.Msg_021;
NETWORK
TITLE = INTERVENTO TERMICO "QF21" ALIM. INVERTER M20 (E3.1)
      AN    "QF21_Inverter_M21";
      S     "DB_OP".Allarmi.Msg_022;
NETWORK
TITLE = INTERVENTO TERMICO "QF22" ALIM. INVERTER M20 (E3.2)
      AN    "QF22_Inverter_M22";
      S     "DB_OP".Allarmi.Msg_023;
NETWORK
TITLE = INTERVENTO TERMICO "QF23" ALIM. INVERTER M20 (E3.3)
      AN    "QF23_Inverter_M23";
      S     "DB_OP".Allarmi.Msg_024;
NETWORK
TITLE = INTERVENTO TERMICO "QF24" ALIM. INVERTER M20 (E3.4)
      AN    "QF24_Inverter_M24";
      S     "DB_OP".Allarmi.Msg_025;
NETWORK
TITLE = INTERVENTO TERMICO "QF25" ALIM. INVERTER M20 (E3.5)
      AN    "QF25_Inverter_M25";
      S     "DB_OP".Allarmi.Msg_026;
NETWORK
TITLE = INTERVENTO TERMICO "QF26" ALIM. INVERTER M20 (E3.6)
      AN    "QF26_Inverter_M26";
      S     "DB_OP".Allarmi.Msg_027;
NETWORK
TITLE = INTERVENTO TERMICO "QF27" ALIM. INVERTER M20 (E3.7)
      AN    "QF27_Inverter_M27";
      S     "DB_OP".Allarmi.Msg_028;
NETWORK
TITLE = INTERVENTO TERMICO "QF28" ALIM. INVERTER M20 (E4.0)
      AN    "QF28_Inverter_M28";
      S     "DB_OP".Allarmi.Msg_029;
NETWORK
TITLE = INTERVENTO TERMICO "QF29" ALIM. INVERTER M20 (E4.1)
      AN    "QF29_Inverter_M29";
      S     "DB_OP".Allarmi.Msg_030;
NETWORK
TITLE = INTERVENTO TERMICO "QF30" ALIM. INVERTER M20 (E4.2)
      AN    "QF30_Inverter_M30";
      S     "DB_OP".Allarmi.Msg_031;
NETWORK
TITLE = INTERVENTO TERMICO "QF31" ALIM. INVERTER M20 (E4.3)
      AN    "QF31_Inverter_M31";
      S     "DB_OP".Allarmi.Msg_032;
NETWORK
TITLE = INTERVENTO TERMICO "QF32" ALIM. INVERTER M20 (E4.4)
      AN    "QF32_Inverter_M32";
      S     "DB_OP".Allarmi.Msg_033;
NETWORK
TITLE = INTERVENTO TERMICO "QF33" ALIM. INVERTER M20 (E4.5)
      AN    "QF33_Inverter_M33";
      S     "DB_OP".Allarmi.Msg_034;
NETWORK
TITLE = INTERVENTO TERMICO "QF34" ALIM. INVERTER M20 (E4.6)
      AN    "QF34_Inverter_M34";
      S     "DB_OP".Allarmi.Msg_035;
NETWORK
TITLE = INTERVENTO TERMICO "QF35" ALIM. INVERTER M20 (E4.7)
      AN    "QF35_Inverter_M35";
      S     "DB_OP".Allarmi.Msg_036;
NETWORK
TITLE = INTERVENTO TERMICO "QF36"(E5.0)
      AN    "QF36_Spare";
      A     "OFF";
      S     "DB_OP".Allarmi.Msg_037;
NETWORK
TITLE = INTERVENTO PROTEZIONE "QF6" VENTILAZIONE QUADRO (E5.1)
      AN    "QF6_Ventilazione_Quadro";
      A     "TODO";
      S     "DB_OP".Allarmi.Msg_041;
NETWORK
TITLE = INTERVENTO PROTEZIONE "QF8"  (E5.2)
      AN    "QF8_Alim_PS_Comandi";
      S     "DB_OP".Allarmi.Msg_042;
NETWORK
TITLE = INTERVENTO PROTEZIONE "QF19" ALIM. CIRCUITI D'EMERGENZA  (E5.3)
      AN    "QF19_Alim_Circuiti_Emerg";
      S     "DB_OP".Allarmi.Msg_043;
NETWORK
TITLE = INTERVENTO PROTEZIONE "QF10" ALIM. COMANDI QUADRO (E5.4)
      AN    "QF10_Alim_Comandi_Quadro";
      S     "DB_OP".Allarmi.Msg_044;
NETWORK
TITLE = INTERVENTO PROTEZIONE "QF11" ALIM. COMANDI JP1  (E5.5)
      AN    "QF11_Alim_Comandi_JP1";
      S     "DB_OP".Allarmi.Msg_045;
NETWORK
TITLE = INTERVENTO PROTEZIONE "QF12" ALIM. COMANDI JP2  (E5.6)
      AN    "QF12_Alim_Comandi_JP2";
      A     "TODO";
      S     "DB_OP".Allarmi.Msg_046;
NETWORK
TITLE = INTERVENTO PROTEZIONE "QF13" ALIM. COMANDI JP3  (E5.7)
      AN    "QF13_Alim_Comandi_JP3";
      A     "TODO";
      S     "DB_OP".Allarmi.Msg_047;
NETWORK
TITLE = FAULT NODO PROFIBUS 3 (INVERTER "M20")
      A     DB125.DBX 1240.2;
      S     "DB_OP".Allarmi.Msg_049;
NETWORK
TITLE = FAULT NODO PROFIBUS 4 (INVERTER "M21")
      A     DB125.DBX 1240.3;
      S     "DB_OP".Allarmi.Msg_050;
NETWORK
TITLE = FAULT NODO PROFIBUS 3 (INVERTER "M20")
      A     DB125.DBX 1240.4;
      S     "DB_OP".Allarmi.Msg_051;
NETWORK
TITLE = FAULT NODO PROFIBUS 3 (INVERTER "M20")
      A     DB125.DBX 1240.5;
      S     "DB_OP".Allarmi.Msg_052;
NETWORK
TITLE = FAULT NODO PROFIBUS 3 (INVERTER "M20")
      A     DB125.DBX 1240.6;
      S     "DB_OP".Allarmi.Msg_053;
NETWORK
TITLE = FAULT NODO PROFIBUS 3 (INVERTER "M20")
      A     DB125.DBX 1240.7;
      S     "DB_OP".Allarmi.Msg_054;
NETWORK
TITLE = FAULT NODO PROFIBUS 9 (INVERTER "M26")
      A     DB125.DBX 1241.0;
      S     "DB_OP".Allarmi.Msg_055;
NETWORK
TITLE = FAULT NODO PROFIBUS 10 (INVERTER "M27")
      A     DB125.DBX 1241.1;
      S     "DB_OP".Allarmi.Msg_056;
NETWORK
TITLE = FAULT NODO PROFIBUS 11 (INVERTER "M28")
      A     DB125.DBX 1241.2;
      S     "DB_OP".Allarmi.Msg_057;
NETWORK
TITLE = FAULT NODO PROFIBUS 12 (INVERTER "M29")
      A     DB125.DBX 1241.3;
      S     "DB_OP".Allarmi.Msg_058;
NETWORK
TITLE = FAULT NODO PROFIBUS 13 (INVERTER "M30")
      A     DB125.DBX 1241.4;
      S     "DB_OP".Allarmi.Msg_059;
NETWORK
TITLE = FAULT NODO PROFIBUS 14 (INVERTER "M31")
      A     DB125.DBX 1241.5;
      S     "DB_OP".Allarmi.Msg_060;
NETWORK
TITLE = FAULT NODO PROFIBUS 15 (INVERTER "M32")
      A     DB125.DBX 1241.6;
      S     "DB_OP".Allarmi.Msg_061;
NETWORK
TITLE = FAULT NODO PROFIBUS 16 (INVERTER "M33")
      A     DB125.DBX 1241.7;
      S     "DB_OP".Allarmi.Msg_062;
NETWORK
TITLE = FAULT NODO PROFIBUS 17 (INVERTER "M34")
      A     DB125.DBX 1242.0;
      S     "DB_OP".Allarmi.Msg_063;
NETWORK
TITLE = FAULT NODO PROFIBUS 18 (INVERTER "M35")
      A     DB125.DBX 1242.1;
      S     "DB_OP".Allarmi.Msg_064;
NETWORK
TITLE = FAULT NODO PROFIBUS 24 (DP/DP COUPLER FORNO)
      A     DB125.DBX 1242.7;
      S     "DB_OP".Allarmi.Msg_065;
NETWORK
TITLE = FAULT NODO PROFIBUS 25 (ET200S - BOX JP1)
      A     DB125.DBX 1243.0;
      L     S5T#2S;
      SF    "T120";
      NOP   0;
      NOP   0;
      NOP   0;
      A     "T120";
      S     "DB_OP".Allarmi.Msg_066;
NETWORK
TITLE = FAULT NODO PROFIBUS 18 (INVERTER "M35")
      A     DB125.DBX 1243.1;
      L     S5T#2S;
      SF    "T121";
      NOP   0;
      NOP   0;
      NOP   0;
      A     "T121";
      S     "DB_OP".Allarmi.Msg_067;
NETWORK
TITLE = FAULT NODO PROFIBUS 27 (ET200S - BOX JP3)
      A     DB125.DBX 1243.2;
      L     S5T#2S;
      SF    "T122";
      NOP   0;
      NOP   0;
      NOP   0;
      A     "T122";
      S     "DB_OP".Allarmi.Msg_068;
NETWORK
TITLE =
      A     "EV_Salita_Traslatore";
      AN    "M130.0";
      L     S5T#20S;
      SD    "T100";
      NOP   0;
      NOP   0;
      NOP   0;
      A     "T100";
      S     "DB_OP".Allarmi.Msg_070;
NETWORK
TITLE =
      A     "EV_Discesa_Traslatore";
      AN    "M130.1";
      L     S5T#10S;
      SD    "T101";
      NOP   0;
      NOP   0;
      NOP   0;
      A     "T101";
      S     "DB_OP".Allarmi.Msg_071;
NETWORK
TITLE =
      A     "EV_Salita_Nastro_Prel_1";
      AN    "M130.2";
      L     S5T#3S;
      SD    "T102";
      NOP   0;
      NOP   0;
      NOP   0;
      A     "T102";
      S     "DB_OP".Allarmi.Msg_072;
NETWORK
TITLE =
      A     "EV_Discesa_Nastro_Prel_1";
      AN    "M130.3";
      L     S5T#3S;
      SD    "T103";
      NOP   0;
      NOP   0;
      NOP   0;
      A     "T103";
      S     "DB_OP".Allarmi.Msg_073;
NETWORK
TITLE =
      A     "EV_Salita_Nastro_Depos_1";
      AN    "M130.4";
      L     S5T#3S;
      SD    "T104";
      NOP   0;
      NOP   0;
      NOP   0;
      A     "T104";
      S     "DB_OP".Allarmi.Msg_074;
NETWORK
TITLE =
      A     "EV_Discesa_Nastro_Depos1";
      AN    "M130.5";
      L     S5T#3S;
      SD    "T105";
      NOP   0;
      NOP   0;
      NOP   0;
      A     "T105";
      S     "DB_OP".Allarmi.Msg_075;
NETWORK
TITLE =
      A     "EV_Salita_Nastro_Prel_2";
      AN    "M130.6";
      L     S5T#3S;
      SD    "T106";
      NOP   0;
      NOP   0;
      NOP   0;
      A     "T106";
      S     "DB_OP".Allarmi.Msg_076;
NETWORK
TITLE =
      A     "EV_Discesa_Nastro_Prel_2";
      AN    "M130.7";
      L     S5T#3S;
      SD    "T107";
      NOP   0;
      NOP   0;
      NOP   0;
      A     "T107";
      S     "DB_OP".Allarmi.Msg_077;
NETWORK
TITLE =
      A     "EV_Salita_Nastro_Depos_2";
      AN    "M131.0";
      L     S5T#3S;
      SD    "T108";
      NOP   0;
      NOP   0;
      NOP   0;
      A     "T108";
      S     "DB_OP".Allarmi.Msg_078;
NETWORK
TITLE =
      A     "EV_Discesa_Nastro_Depos2";
      AN    "M131.1";
      L     S5T#3S;
      SD    "T109";
      NOP   0;
      NOP   0;
      NOP   0;
      A     "T109";
      S     "DB_OP".Allarmi.Msg_079;
NETWORK
TITLE =
      A     "EV_Salita_Nast_Prel_sca1";
      AN    "M131.2";
      L     S5T#3S;
      SD    "T110";
      NOP   0;
      NOP   0;
      NOP   0;
      A     "T110";
      S     "DB_OP".Allarmi.Msg_080;
NETWORK
TITLE =
      A     "EV_Disce_Nast_Prel_sca1";
      AN    "M131.3";
      L     S5T#3S;
      SD    "T111";
      NOP   0;
      NOP   0;
      NOP   0;
      A     "T111";
      S     "DB_OP".Allarmi.Msg_081;
NETWORK
TITLE =
      A     "EV_Salita_Nast_Prel_sca2";
      AN    "M131.4";
      L     S5T#3S;
      SD    "T112";
      NOP   0;
      NOP   0;
      NOP   0;
      A     "T112";
      S     "DB_OP".Allarmi.Msg_082;
NETWORK
TITLE =
      A     "EV_Disce_Nast_Prel_sca2";
      AN    "M131.5";
      L     S5T#3S;
      SD    "T113";
      NOP   0;
      NOP   0;
      NOP   0;
      A     "T113";
      S     "DB_OP".Allarmi.Msg_083;
NETWORK
TITLE = TIMEOUT SENSORE PASSO CADENZATORE INGRESSO LINEA 2 (E24.0)
      A(;
      O     "Comando_M7";
      O     "DB_OP".Allarmi.Msg_084;
      );
      AN    "Proximity_0_Cadenzatore1";
      =     L 0.0;
      A     L 0.0;
      A     "T114";
      S     "DB_OP".Allarmi.Msg_084;
      A     L 0.0;
      BLD   102;
      L     S5T#5S;
      SD    "T114";
NETWORK
TITLE = TIMEOUT SENSORE PASSO CADENZATORE INGRESSO LINEA 1 (E24.1)
      A(;
      O     "Comando_M8";
      O     "DB_OP".Allarmi.Msg_085;
      );
      AN    "Proximity_0_Cadenzatore2";
      =     L 0.0;
      A     L 0.0;
      A     "T115";
      S     "DB_OP".Allarmi.Msg_085;
      A     L 0.0;
      BLD   102;
      L     S5T#5S;
      SD    "T115";
NETWORK
TITLE = TIMEOUT SENSORE PASSO CADENZATORE ACCUMULO "A" LINEA 2 (E27.2)
      A(;
      O     "Comando_M16";
      O     "DB_OP".Allarmi.Msg_086;
      );
      AN    "Proximity_0_Cadenz_scar1";
      =     L 0.0;
      A     L 0.0;
      A     "T116";
      S     "DB_OP".Allarmi.Msg_086;
      A     L 0.0;
      BLD   102;
      L     S5T#6S;
      SD    "T116";
NETWORK
TITLE = TIMEOUT SENSORE PASSO CADENZATORE ACCUMULO "B" LINEA 2 (E27.3)
      A(;
      O     "Comando_M18";
      O     "DB_OP".Allarmi.Msg_087;
      );
      AN    "Proximity_0_Cadenz_scar2";
      =     L 0.0;
      A     L 0.0;
      A     "T117";
      S     "DB_OP".Allarmi.Msg_087;
      A     L 0.0;
      BLD   102;
      L     S5T#6S;
      SD    "T117";
NETWORK
TITLE = CADENZATORE INGRESSO LINEA 2 NON IN FASE (E24.0)
      AN    "Comando_M7";
      AN    "Proximity_0_Cadenzatore1";
      S     "DB_OP".Allarmi.Msg_089;
NETWORK
TITLE = CADENZATORE INGRESSO LINEA 1 NON IN FASE (E24.1)
      AN    "Comando_M8";
      AN    "Proximity_0_Cadenzatore2";
      S     "DB_OP".Allarmi.Msg_090;
NETWORK
TITLE = CADENZATORE ACCUMULO "A" LINEA 2 NON IN FASE (E27.2)
      AN    "Comando_M16";
      AN    "Proximity_0_Cadenz_scar1";
      S     "DB_OP".Allarmi.Msg_091;
NETWORK
TITLE = CADENZATORE ACCUMULO "B" LINEA 2 NON IN FASE (E27.3)
      AN    "Comando_M18";
      AN    "Proximity_0_Cadenz_scar2";
      S     "DB_OP".Allarmi.Msg_092;
NETWORK
TITLE = FOTOCELLULA ARRESTO PACCO 4 FILE TRASLATORE E' RIMASTA IMPEGNATA
      A     "TODO";
      A     "IR_Stop_Traslazione";
      S     "DB_OP".Allarmi.Msg_093;
NETWORK
TITLE = FOTOCELLULA ARRESTO PACCO 4 FILE DAVANTI LINEA 2 E' RIMASTA IMPE
      A     "TODO";
      S     "DB_OP".Allarmi.Msg_094;
NETWORK
TITLE = FOTOCELLULA ARRESTO PACCO 4 FILE DAVANTI LINEA 1 E' RIMASTA IMPE
      A     "TODO";
      S     "DB_OP".Allarmi.Msg_095;
NETWORK
TITLE = FOTOCELLULA ARRESTO BARRA DAVANTI CADENZATORE LINEA 2 E' RIMASTA
      A     "TODO";
      S     "DB_OP".Allarmi.Msg_096;
NETWORK
TITLE = FOTOCELLULA ARRESTO BARRA DAVANTI CADENZATORE LINEA 1 E' RIMASTA
      A     "TODO";
      S     "DB_OP".Allarmi.Msg_097;
NETWORK
TITLE = FOTOCELLULA ARRESTO BARRA SU RULLIERA 1 INGRESSO ESTR. LINEA 2 E
      A     "TODO";
      S     "DB_OP".Allarmi.Msg_098;
NETWORK
TITLE = FOTOCELLULA ARRESTO BARRA SU RULLIERA 1 INGRESSO ESTR. LINEA 1 E
      A     "TODO";
      S     "DB_OP".Allarmi.Msg_099;
NETWORK
TITLE = FOTOCELLULA ARRESTO BARRA SU CADENZATORE ACCUMULO "A" LINEA 2 E'
      A     "TODO";
      S     "DB_OP".Allarmi.Msg_100;
NETWORK
TITLE = FOTOCELLULA ARRESTO BARRA SU CADENZATORE ACCUMULO "B" LINEA 2 E'
      A     "TODO";
      S     "DB_OP".Allarmi.Msg_101;
NETWORK
TITLE = FOTOCELLULA ARRESTO BARRA SU DEVIATORE ACCUMULO "A" LINEA 1 E' R
      A     "TODO";
      S     "DB_OP".Allarmi.Msg_102;
NETWORK
TITLE = FOTOCELLULA ARRESTO BARRA SU DEVIATORE ACCUMULO "B" LINEA 1 E' R
      A     "TODO";
      S     "DB_OP".Allarmi.Msg_103;
NETWORK
TITLE = TIMEOUT CICLO TRASFERITORE O MANCATA LETTURA FOTOCELLULA ARRESTO
      A     "TODO";
      S     "DB_OP".Allarmi.Msg_105;
NETWORK
TITLE = TIMEOUT CICLO TRASFERIMENTO 4 BARRE VERSO LINEA 2 O MANCATA LETT
      A     "TODO";
      S     "DB_OP".Allarmi.Msg_106;
NETWORK
TITLE = TIMEOUT CICLO TRASFERIMENTO 4 BARRE VERSO LINEA 1 O MANCATA LETT
      A     "TODO";
      S     "DB_OP".Allarmi.Msg_107;
NETWORK
TITLE = TIMEOUT CICLO ALIMENTAZIONE CADENZATORE LINEA 2 O MANCATA LETTUR
      A     "TODO";
      S     "DB_OP".Allarmi.Msg_108;
NETWORK
TITLE = TIMEOUT CICLO ALIMENTAZIONE CADENZATORE LINEA 1 O MANCATA LETTUR
      A     "TODO";
      S     "DB_OP".Allarmi.Msg_109;
NETWORK
TITLE = LINEA ACCUMULO "A" INFERIORE PIENA
      A     "M44.1";
      A     "IR_Stop_Banco2_Scaric_L";
      =     "DB_OP".Allarmi.Msg_110;
NETWORK
TITLE = LINEA ACCUMULO "A" SUPERIORE PIENA
      A     "M24.6";
      A     "IR_Stop_Banco1_Scaric_H";
      =     "DB_OP".Allarmi.Msg_111;
NETWORK
TITLE = LINEA ACCUMULO "B" INFERIORE PIENA
      A     "M45.4";
      A     "IR_Stop_Banco1_Scaric_L";
      =     "DB_OP".Allarmi.Msg_112;
NETWORK
TITLE = LINEA ACCUMULO "B" SUPERIORE PIENA 
      A     "M26.4";
      A     "IR_Stop_Banco2_Scaric_H";
      =     "DB_OP".Allarmi.Msg_113;
NETWORK
TITLE = INVERTER A1 MOTORE "M20" IN ALLARME
      A     "M66.0";
      S     "DB_OP".Allarmi.Msg_114;
NETWORK
TITLE = INVERTER A2 MOTORE "M21" IN ALLARME
      A     "M66.1";
      S     "DB_OP".Allarmi.Msg_115;
NETWORK
TITLE = INVERTER A3 MOTORE "M22" IN ALLARME
      A     "M66.2";
      S     "DB_OP".Allarmi.Msg_116;
NETWORK
TITLE = INVERTER A2 MOTORE "M21" IN ALLARME
      A     "M66.3";
      S     "DB_OP".Allarmi.Msg_117;
NETWORK
TITLE = INVERTER A5 MOTORE "M24" IN ALLARME
      A     "M66.4";
      S     "DB_OP".Allarmi.Msg_118;
NETWORK
TITLE = INVERTER A6 MOTORE "M25" IN ALLARME
      A     "M66.5";
      S     "DB_OP".Allarmi.Msg_119;
NETWORK
TITLE = INVERTER A7 MOTORE "M26" IN ALLARME
      A     "M66.6";
      S     "DB_OP".Allarmi.Msg_120;
NETWORK
TITLE = INVERTER A8 MOTORE "M27" IN ALLARME
      A     "M66.7";
      S     "DB_OP".Allarmi.Msg_121;
NETWORK
TITLE = INVERTER A9 MOTORE "M28" IN ALLARME
      A     "M67.0";
      S     "DB_OP".Allarmi.Msg_122;
NETWORK
TITLE = INVERTER A10 MOTORE "M29" IN ALLARME
      A     "M67.1";
      S     "DB_OP".Allarmi.Msg_123;
NETWORK
TITLE = INVERTER A11 MOTORE "M30" IN ALLARME
      A     "M67.2";
      S     "DB_OP".Allarmi.Msg_124;
NETWORK
TITLE = INVERTER A12 MOTORE "M31" IN ALLARME
      A     "M67.3";
      S     "DB_OP".Allarmi.Msg_125;
NETWORK
TITLE = INVERTER A13 MOTORE "M32" IN ALLARME
      A     "M67.4";
      S     "DB_OP".Allarmi.Msg_126;
NETWORK
TITLE = INVERTER A14 MOTORE "M33" IN ALLARME
      A     "M67.5";
      S     "DB_OP".Allarmi.Msg_127;
NETWORK
TITLE = INVERTER A15 MOTORE "M34" IN ALLARME
      A     "M67.6";
      S     "DB_OP".Allarmi.Msg_128;
NETWORK
TITLE = INVERTER A16 MOTORE "M35" IN ALLARME
      A     "M67.7";
      S     "DB_OP".Allarmi.Msg_129;
NETWORK
TITLE =
      CALL  "FC_AllarmeAttivo" (
           RET_VAL                  := "ALLARME",
           Allarmi                  := "DB_OP".Allarmi);
      NOP   0;
NETWORK
TITLE = MOTORE M1 IN ALLARME
      O     "DB_OP".Allarmi.Msg_001;
      O     "DB_OP".Allarmi.Msg_045;
      =     "M70.0";
NETWORK
TITLE = MOTORE M2 IN ALLARME
      O     "DB_OP".Allarmi.Msg_002;
      O     "DB_OP".Allarmi.Msg_045;
      =     "M70.1";
NETWORK
TITLE = MOTORE M3 IN ALLARME
      O     "DB_OP".Allarmi.Msg_003;
      O     "DB_OP".Allarmi.Msg_066;
      O     "DB_OP".Allarmi.Msg_045;
      O     "DB_OP".Allarmi.Msg_070;
      O     "DB_OP".Allarmi.Msg_071;
      =     "M70.2";
NETWORK
TITLE = MOTORE M4 IN ALLARME
      O     "DB_OP".Allarmi.Msg_004;
      O     "DB_OP".Allarmi.Msg_067;
      O     "DB_OP".Allarmi.Msg_072;
      O     "DB_OP".Allarmi.Msg_073;
      =     "M70.3";
NETWORK
TITLE = MOTORE M5 IN ALLARME
      O     "DB_OP".Allarmi.Msg_005;
      O     "DB_OP".Allarmi.Msg_067;
      O     "DB_OP".Allarmi.Msg_084;
      O     "DB_OP".Allarmi.Msg_089;
      =     "M70.4";
NETWORK
TITLE = MOTORE M6 IN ALLARME
      O     "DB_OP".Allarmi.Msg_006;
      O     "DB_OP".Allarmi.Msg_067;
      O     "DB_OP".Allarmi.Msg_074;
      O     "DB_OP".Allarmi.Msg_075;
      =     "M70.5";
NETWORK
TITLE = MOTORE M7 IN ALLARME
      O     "DB_OP".Allarmi.Msg_007;
      O     "DB_OP".Allarmi.Msg_067;
      O     "DB_OP".Allarmi.Msg_084;
      O     "DB_OP".Allarmi.Msg_089;
      =     "M70.6";
NETWORK
TITLE = MOTORE M8 IN ALLARME
      O     "DB_OP".Allarmi.Msg_008;
      O     "DB_OP".Allarmi.Msg_067;
      O     "DB_OP".Allarmi.Msg_085;
      O     "DB_OP".Allarmi.Msg_090;
      =     "M70.7";
NETWORK
TITLE = MOTORE M9 IN ALLARME
      O     "DB_OP".Allarmi.Msg_009;
      O     "DB_OP".Allarmi.Msg_067;
      O     "DB_OP".Allarmi.Msg_078;
      O     "DB_OP".Allarmi.Msg_079;
      =     "M71.0";
NETWORK
TITLE = MOTORE M10 IN ALLARME
      O     "DB_OP".Allarmi.Msg_010;
      O     "DB_OP".Allarmi.Msg_067;
      O     "DB_OP".Allarmi.Msg_085;
      O     "DB_OP".Allarmi.Msg_090;
      =     "M71.1";
NETWORK
TITLE = MOTORE M11 IN ALLARME
      O     "DB_OP".Allarmi.Msg_011;
      O     "DB_OP".Allarmi.Msg_067;
      O     "DB_OP".Allarmi.Msg_076;
      O     "DB_OP".Allarmi.Msg_077;
      =     "M71.2";
NETWORK
TITLE = MOTORE M12 IN ALLARME
      O     "DB_OP".Allarmi.Msg_012;
      O     "DB_OP".Allarmi.Msg_068;
      O     "DB_OP".Allarmi.Msg_080;
      O     "DB_OP".Allarmi.Msg_081;
      =     "M71.3";
NETWORK
TITLE = MOTORE M13 IN ALLARME
      O     "DB_OP".Allarmi.Msg_013;
      O     "DB_OP".Allarmi.Msg_068;
      =     "M71.4";
NETWORK
TITLE = MOTORE M14 IN ALLARME
      O     "DB_OP".Allarmi.Msg_014;
      O     "DB_OP".Allarmi.Msg_068;
      O     "DB_OP".Allarmi.Msg_082;
      O     "DB_OP".Allarmi.Msg_083;
      =     "M71.5";
NETWORK
TITLE = MOTORE M15 IN ALLARME
      O     "DB_OP".Allarmi.Msg_015;
      O     "DB_OP".Allarmi.Msg_068;
      =     "M71.6";
NETWORK
TITLE = MOTORE M16 IN ALLARME
      O     "DB_OP".Allarmi.Msg_016;
      O     "DB_OP".Allarmi.Msg_068;
      O     "DB_OP".Allarmi.Msg_086;
      O     "DB_OP".Allarmi.Msg_091;
      =     "M71.7";
NETWORK
TITLE = MOTORE M17 IN ALLARME
      O     "DB_OP".Allarmi.Msg_017;
      O     "DB_OP".Allarmi.Msg_068;
      =     "M72.0";
NETWORK
TITLE = MOTORE M18 IN ALLARME
      O     "DB_OP".Allarmi.Msg_018;
      O     "DB_OP".Allarmi.Msg_068;
      O     "DB_OP".Allarmi.Msg_087;
      O     "DB_OP".Allarmi.Msg_092;
      =     "M72.1";
NETWORK
TITLE = MOTORE M19 IN ALLARME
      O     "DB_OP".Allarmi.Msg_019;
      O     "DB_OP".Allarmi.Msg_068;
      =     "M72.2";
NETWORK
TITLE = MOTORE M20 IN ALLARME
      O     "DB_OP".Allarmi.Msg_021;
      O     "DB_OP".Allarmi.Msg_066;
      O     "DB_OP".Allarmi.Msg_049;
      O     "DB_OP".Allarmi.Msg_114;
      O     "DB_OP".Allarmi.Msg_070;
      O     "DB_OP".Allarmi.Msg_071;
      =     "M72.3";
NETWORK
TITLE = MOTORE M21 IN ALLARME
      O     "DB_OP".Allarmi.Msg_022;
      O     "DB_OP".Allarmi.Msg_050;
      O     "DB_OP".Allarmi.Msg_115;
      =     "M72.4";
NETWORK
TITLE = MOTORE M22 IN ALLARME
      O     "DB_OP".Allarmi.Msg_023;
      O     "DB_OP".Allarmi.Msg_067;
      O     "DB_OP".Allarmi.Msg_051;
      O     "DB_OP".Allarmi.Msg_116;
      O     "DB_OP".Allarmi.Msg_072;
      O     "DB_OP".Allarmi.Msg_073;
      =     "M72.5";
NETWORK
TITLE = MOTORE M23 IN ALLARME
      O     "DB_OP".Allarmi.Msg_024;
      O     "DB_OP".Allarmi.Msg_067;
      O     "DB_OP".Allarmi.Msg_052;
      O     "DB_OP".Allarmi.Msg_117;
      =     "M72.6";
NETWORK
TITLE = MOTORE M24 IN ALLARME
      O     "DB_OP".Allarmi.Msg_025;
      O     "DB_OP".Allarmi.Msg_067;
      O     "DB_OP".Allarmi.Msg_053;
      O     "DB_OP".Allarmi.Msg_118;
      O     "DB_OP".Allarmi.Msg_076;
      O     "DB_OP".Allarmi.Msg_077;
      =     "M72.7";
NETWORK
TITLE = MOTORE M25 IN ALLARME
      O     "DB_OP".Allarmi.Msg_026;
      O     "DB_OP".Allarmi.Msg_067;
      O     "DB_OP".Allarmi.Msg_054;
      O     "DB_OP".Allarmi.Msg_119;
      O     "DB_OP".Allarmi.Msg_074;
      O     "DB_OP".Allarmi.Msg_075;
      =     "M73.0";
NETWORK
TITLE = MOTORE M26 IN ALLARME
      O     "DB_OP".Allarmi.Msg_027;
      O     "DB_OP".Allarmi.Msg_067;
      O     "DB_OP".Allarmi.Msg_055;
      O     "DB_OP".Allarmi.Msg_120;
      =     "M73.1";
NETWORK
TITLE = MOTORE M27 IN ALLARME
      O     "DB_OP".Allarmi.Msg_028;
      O     "DB_OP".Allarmi.Msg_067;
      O     "DB_OP".Allarmi.Msg_056;
      O     "DB_OP".Allarmi.Msg_121;
      O     "DB_OP".Allarmi.Msg_078;
      O     "DB_OP".Allarmi.Msg_079;
      =     "M73.2";
NETWORK
TITLE = MOTORE M28 IN ALLARME
      O     "DB_OP".Allarmi.Msg_029;
      O     "DB_OP".Allarmi.Msg_067;
      O     "DB_OP".Allarmi.Msg_057;
      O     "DB_OP".Allarmi.Msg_122;
      =     "M73.3";
NETWORK
TITLE = MOTORE M29 IN ALLARME
      O     "DB_OP".Allarmi.Msg_030;
      O     "DB_OP".Allarmi.Msg_067;
      O     "DB_OP".Allarmi.Msg_058;
      O     "DB_OP".Allarmi.Msg_123;
      =     "M73.4";
NETWORK
TITLE = MOTORE M30 IN ALLARME
      O     "DB_OP".Allarmi.Msg_031;
      O     "DB_OP".Allarmi.Msg_068;
      O     "DB_OP".Allarmi.Msg_059;
      O     "DB_OP".Allarmi.Msg_124;
      O     "DB_OP".Allarmi.Msg_086;
      O     "DB_OP".Allarmi.Msg_091;
      =     "M73.5";
NETWORK
TITLE = MOTORE M31 IN ALLARME
      O     "DB_OP".Allarmi.Msg_032;
      O     "DB_OP".Allarmi.Msg_068;
      O     "DB_OP".Allarmi.Msg_060;
      O     "DB_OP".Allarmi.Msg_125;
      O     "DB_OP".Allarmi.Msg_087;
      O     "DB_OP".Allarmi.Msg_092;
      =     "M73.6";
NETWORK
TITLE = MOTORE M32 IN ALLARME
      O     "DB_OP".Allarmi.Msg_033;
      O     "DB_OP".Allarmi.Msg_068;
      O     "DB_OP".Allarmi.Msg_061;
      O     "DB_OP".Allarmi.Msg_126;
      =     "M73.7";
NETWORK
TITLE = MOTORE M33 IN ALLARME
      O     "DB_OP".Allarmi.Msg_034;
      O     "DB_OP".Allarmi.Msg_068;
      O     "DB_OP".Allarmi.Msg_062;
      O     "DB_OP".Allarmi.Msg_127;
      O     "DB_OP".Allarmi.Msg_080;
      O     "DB_OP".Allarmi.Msg_081;
      =     "M74.0";
NETWORK
TITLE = MOTORE M34 IN ALLARME
      O     "DB_OP".Allarmi.Msg_035;
      O     "DB_OP".Allarmi.Msg_068;
      O     "DB_OP".Allarmi.Msg_063;
      O     "DB_OP".Allarmi.Msg_128;
      O     "DB_OP".Allarmi.Msg_082;
      O     "DB_OP".Allarmi.Msg_083;
      =     "M74.1";
NETWORK
TITLE = MOTORE M35 IN ALLARME
      O     "DB_OP".Allarmi.Msg_036;
      O     "DB_OP".Allarmi.Msg_064;
      O     "DB_OP".Allarmi.Msg_129;
      =     "M74.2";
NETWORK
TITLE =
NETWORK
TITLE = NODO JP1 ET200S OK
      AN    "DB_OP".Allarmi.Msg_066;
      AN    "DB_OP".Allarmi.Msg_045;
      =     "M74.3";
NETWORK
TITLE = NODO JP2 ET200S OK
      AN    "DB_OP".Allarmi.Msg_067;
      AN    "DB_OP".Allarmi.Msg_046;
      =     "M74.4";
NETWORK
TITLE = NODO JP3 ET200S OK
      AN    "DB_OP".Allarmi.Msg_068;
      AN    "DB_OP".Allarmi.Msg_047;
      =     "M74.5";
END_FUNCTION

FUNCTION "Segnalazioni" : VOID	// FC 2
NAME : Warning
VERSION : 0.1
BEGIN
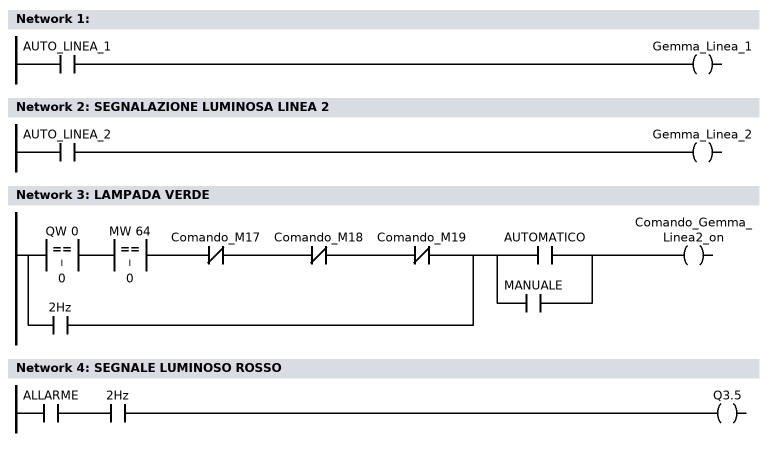
NETWORK
TITLE =
      A     "AUTO_LINEA_1";
      =     "Gemma_Linea_1";
NETWORK
TITLE = SEGNALAZIONE LUMINOSA LINEA 2
      A     "AUTO_LINEA_2";
      =     "Gemma_Linea_2";
NETWORK
TITLE = LAMPADA VERDE
      A(;
      A(;
      L     QW 0;
      L     0;
      ==I;
      );
      A(;
      L     MW 64;
      L     0;
      ==I;
      );
      AN    "Comando_M17";
      AN    "Comando_M18";
      AN    "Comando_M19";
      O     "2Hz";
      );
      A(;
      O     "AUTOMATICO";
      O     "MANUALE";
      );
      =     "Comando_Gemma_Linea2_on";
NETWORK
TITLE = SEGNALE LUMINOSO ROSSO
      A     "ALLARME";
      A     "2Hz";
      =     "Q3.5";
END_FUNCTION

FUNCTION "Consensi Generali" : VOID	// FC 3
NAME : Consensi
VERSION : 0.1
BEGIN
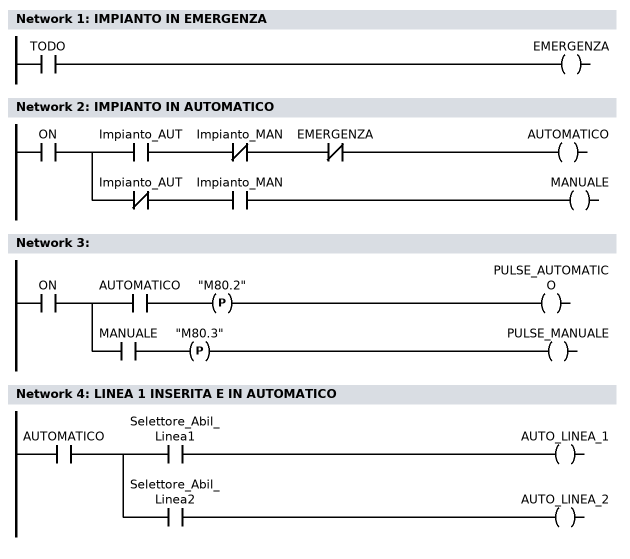
NETWORK
TITLE = IMPIANTO IN EMERGENZA
      A     "TODO";
      =     "EMERGENZA";
NETWORK
TITLE = IMPIANTO IN AUTOMATICO
      A     "ON";
      =     L 0.0;
      A     L 0.0;
      A     "Impianto_AUT";
      AN    "Impianto_MAN";
      AN    "EMERGENZA";
      =     "AUTOMATICO";
      A     L 0.0;
      AN    "Impianto_AUT";
      A     "Impianto_MAN";
      =     "MANUALE";
NETWORK
TITLE =
      A     "ON";
      =     L 0.0;
      A     L 0.0;
      A     "AUTOMATICO";
      FP    "M80.2";
      =     "PULSE_AUTOMATICO";
      A     L 0.0;
      A     "MANUALE";
      FP    "M80.3";
      =     "PULSE_MANUALE";
NETWORK
TITLE = LINEA 1 INSERITA E IN AUTOMATICO
      A     "AUTOMATICO";
      =     L 0.0;
      A     L 0.0;
      A     "Selettore_Abil_Linea1";
      =     "AUTO_LINEA_1";
      A     L 0.0;
      A     "Selettore_Abil_Linea2";
      =     "AUTO_LINEA_2";
END_FUNCTION

FUNCTION "Automatico_zona_ingresso" : VOID	// FC 4
NAME : Auto_In
VERSION : 0.1
BEGIN
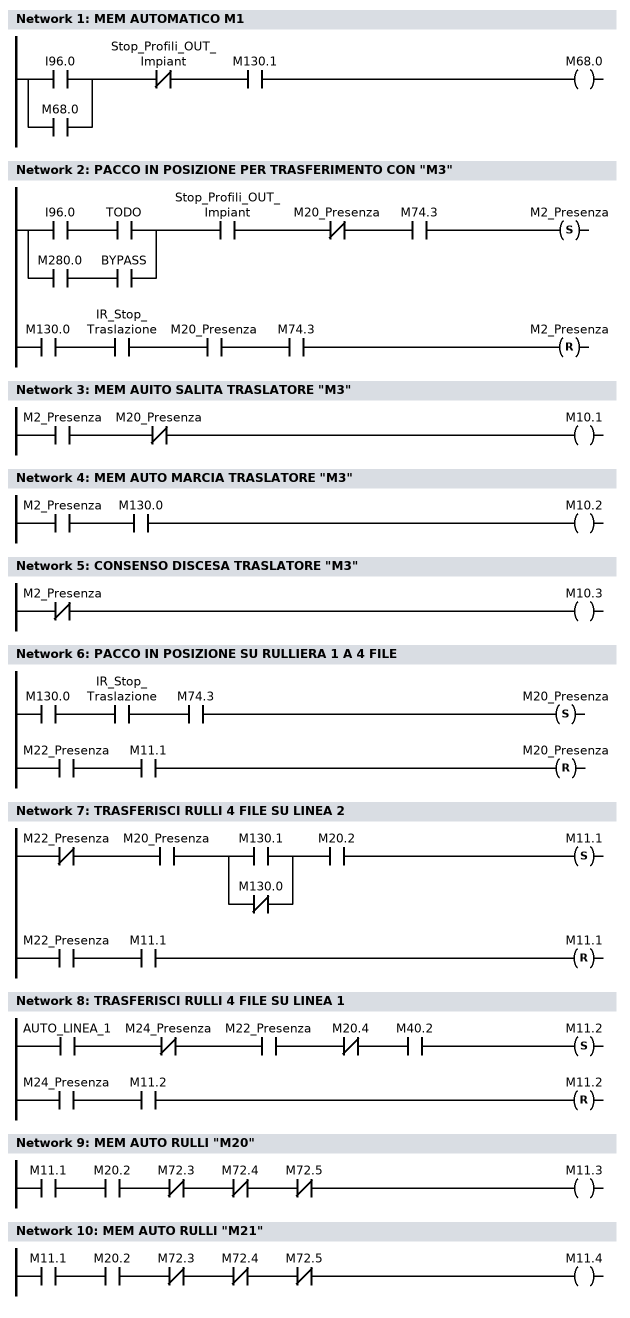
NETWORK
TITLE = MEM AUTOMATICO M1
      A(;
      O     "I96.0";
      O     "M68.0";
      );
      AN    "Stop_Profili_OUT_Impiant";
      A     "M130.1";
      =     "M68.0";
NETWORK
TITLE = PACCO IN POSIZIONE PER TRASFERIMENTO CON "M3"
      A(;
      A     "I96.0";
      A     "TODO";
      O;
      A     "M280.0";
      A     "BYPASS";
      );
      A     "Stop_Profili_OUT_Impiant";
      AN    "M20_Presenza";
      A     "M74.3";
      S     "M2_Presenza";
      A     "M130.0";
      A     "IR_Stop_Traslazione";
      A     "M20_Presenza";
      A     "M74.3";
      R     "M2_Presenza";
      NOP   0;
NETWORK
TITLE = MEM AUITO SALITA TRASLATORE "M3"
      A     "M2_Presenza";
      AN    "M20_Presenza";
      =     "M10.1";
NETWORK
TITLE = MEM AUTO MARCIA TRASLATORE "M3"
      A     "M2_Presenza";
      A     "M130.0";
      =     "M10.2";
NETWORK
TITLE = CONSENSO DISCESA TRASLATORE "M3"
      AN    "M2_Presenza";
      =     "M10.3";
NETWORK
TITLE = PACCO IN POSIZIONE SU RULLIERA 1 A 4 FILE
      A     "M130.0";
      A     "IR_Stop_Traslazione";
      A     "M74.3";
      S     "M20_Presenza";
      A     "M22_Presenza";
      A     "M11.1";
      R     "M20_Presenza";
      NOP   0;
NETWORK
TITLE = TRASFERISCI RULLI 4 FILE SU LINEA 2
      AN    "M22_Presenza";
      A     "M20_Presenza";
      A(;
      O     "M130.1";
      ON    "M130.0";
      );
      A     "M20.2";
      S     "M11.1";
      A     "M22_Presenza";
      A     "M11.1";
      R     "M11.1";
      NOP   0;
NETWORK
TITLE = TRASFERISCI RULLI 4 FILE SU LINEA 1
      A     "AUTO_LINEA_1";
      AN    "M24_Presenza";
      A     "M22_Presenza";
      AN    "M20.4";
      A     "M40.2";
      S     "M11.2";
      A     "M24_Presenza";
      A     "M11.2";
      R     "M11.2";
      NOP   0;
NETWORK
TITLE = MEM AUTO RULLI "M20"
      A     "M11.1";
      A     "M20.2";
      AN    "M72.3";
      AN    "M72.4";
      AN    "M72.5";
      =     "M11.3";
NETWORK
TITLE = MEM AUTO RULLI "M21"
      A     "M11.1";
      A     "M20.2";
      AN    "M72.3";
      AN    "M72.4";
      AN    "M72.5";
      =     "M11.4";
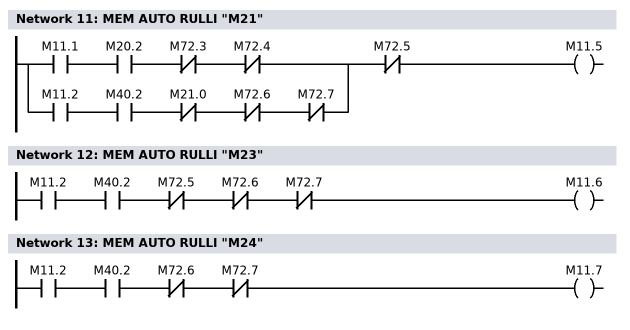
NETWORK
TITLE = MEM AUTO RULLI "M21"
      A(;
      A     "M11.1";
      A     "M20.2";
      AN    "M72.3";
      AN    "M72.4";
      O;
      A     "M11.2";
      A     "M40.2";
      AN    "M21.0";
      AN    "M72.6";
      AN    "M72.7";
      );
      AN    "M72.5";
      =     "M11.5";
NETWORK
TITLE = MEM AUTO RULLI "M23"
      A     "M11.2";
      A     "M40.2";
      AN    "M72.5";
      AN    "M72.6";
      AN    "M72.7";
      =     "M11.6";
NETWORK
TITLE = MEM AUTO RULLI "M24"
      A     "M11.2";
      A     "M40.2";
      AN    "M72.6";
      AN    "M72.7";
      =     "M11.7";
END_FUNCTION

FUNCTION "Automatico_linea_1" : VOID	// FC 5
NAME : Auto_L1
VERSION : 0.1
BEGIN
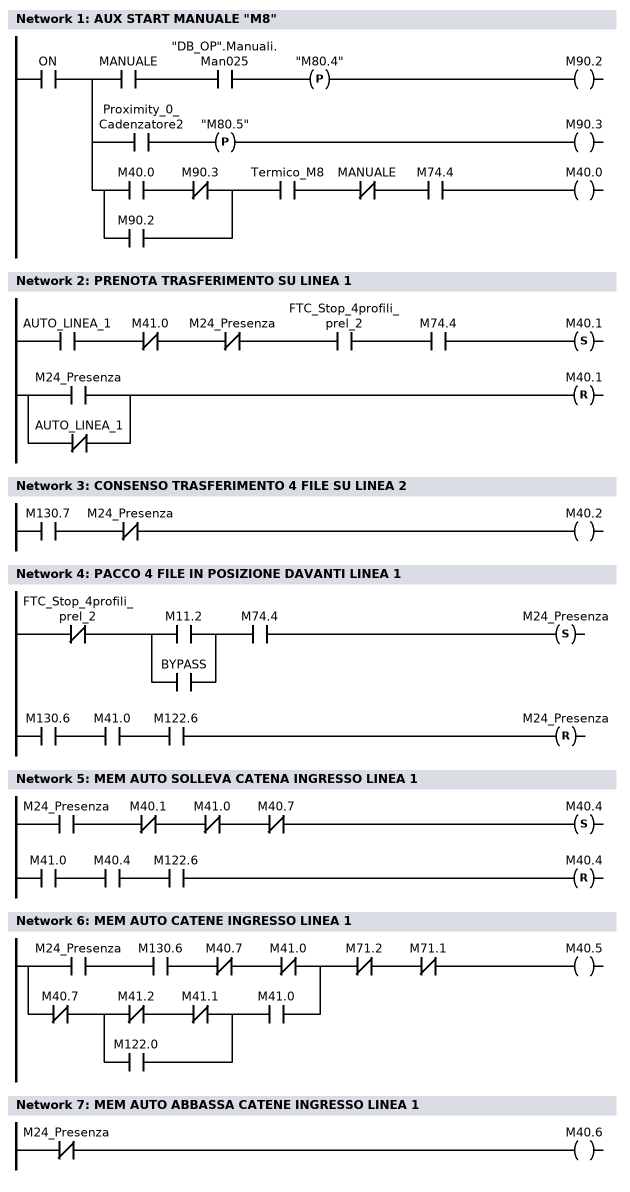
NETWORK
TITLE = AUX START MANUALE "M8"
      A     "ON";
      =     L 0.0;
      A     L 0.0;
      A     "MANUALE";
      A     "DB_OP".Manuali.Man025;
      FP    "M80.4";
      =     "M90.2";
      A     L 0.0;
      A     "Proximity_0_Cadenzatore2";
      FP    "M80.5";
      =     "M90.3";
      A     L 0.0;
      A(;
      A     "M40.0";
      AN    "M90.3";
      O     "M90.2";
      );
      A     "Termico_M8";
      AN    "MANUALE";
      A     "M74.4";
      =     "M40.0";
NETWORK
TITLE = PRENOTA TRASFERIMENTO SU LINEA 1
      A     "AUTO_LINEA_1";
      AN    "M41.0";
      AN    "M24_Presenza";
      A     "FTC_Stop_4profili_prel_2";
      A     "M74.4";
      S     "M40.1";
      A(;
      O     "M24_Presenza";
      ON    "AUTO_LINEA_1";
      );
      R     "M40.1";
      NOP   0;
NETWORK
TITLE = CONSENSO TRASFERIMENTO 4 FILE SU LINEA 2
      A     "M130.7";
      AN    "M24_Presenza";
      =     "M40.2";
NETWORK
TITLE = PACCO 4 FILE IN POSIZIONE DAVANTI LINEA 1
      AN    "FTC_Stop_4profili_prel_2";
      A(;
      O     "M11.2";
      O     "BYPASS";
      );
      A     "M74.4";
      S     "M24_Presenza";
      A     "M130.6";
      A     "M41.0";
      A     "M122.6";
      R     "M24_Presenza";
      NOP   0;
NETWORK
TITLE = MEM AUTO SOLLEVA CATENA INGRESSO LINEA 1
      A     "M24_Presenza";
      AN    "M40.1";
      AN    "M41.0";
      AN    "M40.7";
      S     "M40.4";
      A     "M41.0";
      A     "M40.4";
      A     "M122.6";
      R     "M40.4";
      NOP   0;
NETWORK
TITLE = MEM AUTO CATENE INGRESSO LINEA 1
      A(;
      A     "M24_Presenza";
      A     "M130.6";
      AN    "M40.7";
      AN    "M41.0";
      O;
      AN    "M40.7";
      A(;
      AN    "M41.2";
      AN    "M41.1";
      O     "M122.0";
      );
      A     "M41.0";
      );
      AN    "M71.2";
      AN    "M71.1";
      =     "M40.5";
NETWORK
TITLE = MEM AUTO ABBASSA CATENE INGRESSO LINEA 1
      AN    "M24_Presenza";
      =     "M40.6";
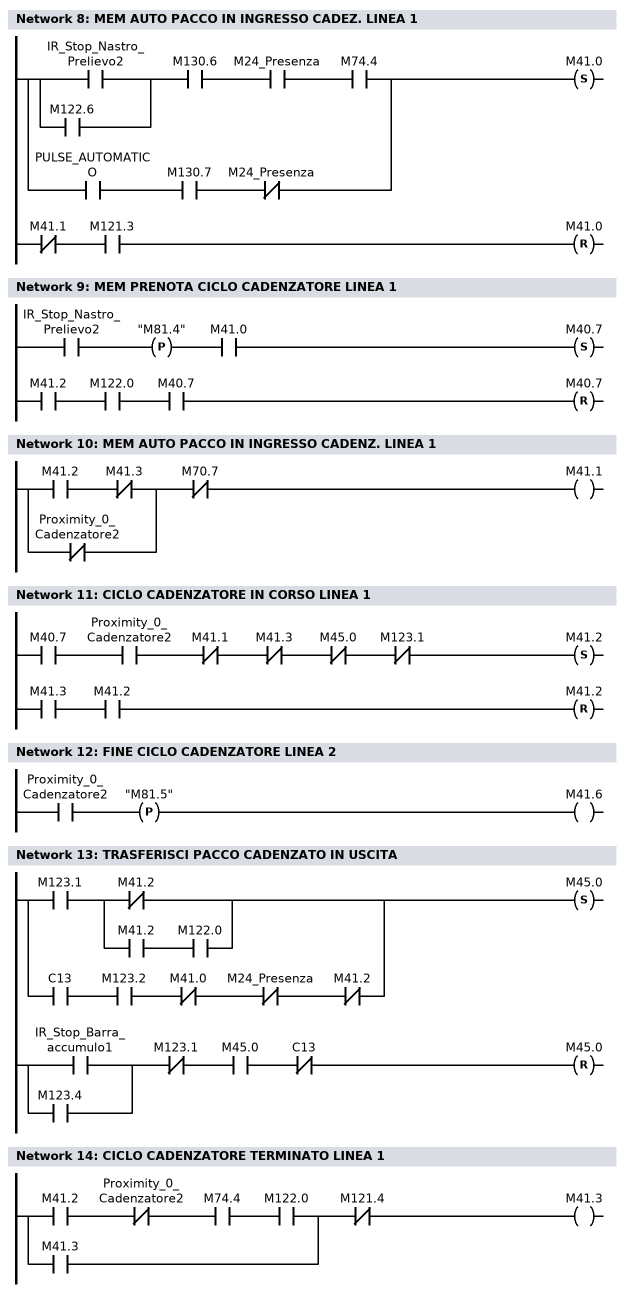
NETWORK
TITLE = MEM AUTO PACCO IN INGRESSO CADEZ. LINEA 1
      A(;
      A(;
      O     "IR_Stop_Nastro_Prelievo2";
      O     "M122.6";
      );
      A     "M130.6";
      A     "M24_Presenza";
      A     "M74.4";
      O;
      A     "PULSE_AUTOMATICO";
      A     "M130.7";
      AN    "M24_Presenza";
      );
      S     "M41.0";
      AN    "M41.1";
      A     "M121.3";
      R     "M41.0";
      NOP   0;
NETWORK
TITLE = MEM PRENOTA CICLO CADENZATORE LINEA 1
      A     "IR_Stop_Nastro_Prelievo2";
      FP    "M81.4";
      A     "M41.0";
      S     "M40.7";
      A     "M41.2";
      A     "M122.0";
      A     "M40.7";
      R     "M40.7";
      NOP   0;
NETWORK
TITLE = MEM AUTO PACCO IN INGRESSO CADENZ. LINEA 1
      A(;
      A     "M41.2";
      AN    "M41.3";
      ON    "Proximity_0_Cadenzatore2";
      );
      AN    "M70.7";
      =     "M41.1";
NETWORK
TITLE = CICLO CADENZATORE IN CORSO LINEA 1
      A     "M40.7";
      A     "Proximity_0_Cadenzatore2";
      AN    "M41.1";
      AN    "M41.3";
      AN    "M45.0";
      AN    "M123.1";
      S     "M41.2";
      A     "M41.3";
      A     "M41.2";
      R     "M41.2";
      NOP   0;
NETWORK
TITLE = FINE CICLO CADENZATORE LINEA 2
      A     "Proximity_0_Cadenzatore2";
      FP    "M81.5";
      =     "M41.6";
NETWORK
TITLE = TRASFERISCI PACCO CADENZATO IN USCITA
      A(;
      A     "M123.1";
      A(;
      ON    "M41.2";
      O;
      A     "M41.2";
      A     "M122.0";
      );
      O;
      A     "C13";
      A     "M123.2";
      AN    "M41.0";
      AN    "M24_Presenza";
      AN    "M41.2";
      );
      S     "M45.0";
      A(;
      O     "IR_Stop_Barra_accumulo1";
      O     "M123.4";
      );
      AN    "M123.1";
      A     "M45.0";
      AN    "C13";
      R     "M45.0";
      NOP   0;
NETWORK
TITLE = CICLO CADENZATORE TERMINATO LINEA 1
      A(;
      A     "M41.2";
      AN    "Proximity_0_Cadenzatore2";
      A     "M74.4";
      A     "M122.0";
      O     "M41.3";
      );
      AN    "M121.4";
      =     "M41.3";
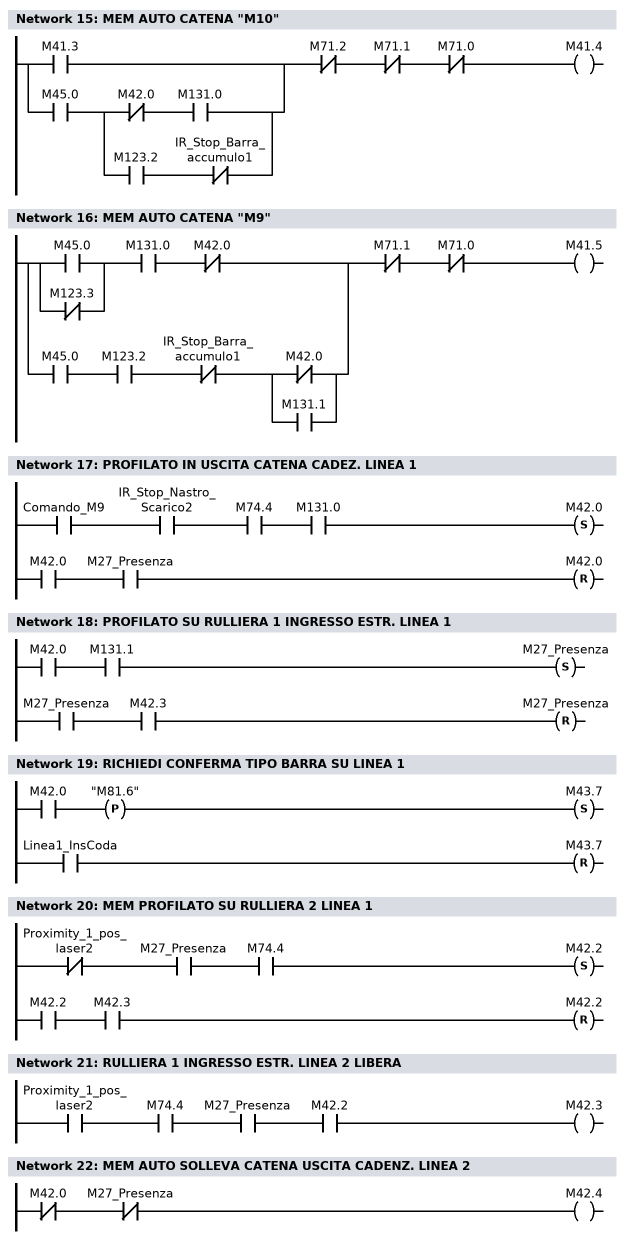
NETWORK
TITLE = MEM AUTO CATENA "M10"
      A(;
      O     "M41.3";
      O;
      A     "M45.0";
      A(;
      AN    "M42.0";
      A     "M131.0";
      O;
      A     "M123.2";
      AN    "IR_Stop_Barra_accumulo1";
      );
      );
      AN    "M71.2";
      AN    "M71.1";
      AN    "M71.0";
      =     "M41.4";
NETWORK
TITLE = MEM AUTO CATENA "M9"
      A(;
      A(;
      O     "M45.0";
      ON    "M123.3";
      );
      A     "M131.0";
      AN    "M42.0";
      O;
      A     "M45.0";
      A     "M123.2";
      AN    "IR_Stop_Barra_accumulo1";
      A(;
      ON    "M42.0";
      O     "M131.1";
      );
      );
      AN    "M71.1";
      AN    "M71.0";
      =     "M41.5";
NETWORK
TITLE = PROFILATO IN USCITA CATENA CADEZ. LINEA 1
      A     "Comando_M9";
      A     "IR_Stop_Nastro_Scarico2";
      A     "M74.4";
      A     "M131.0";
      S     "M42.0";
      A     "M42.0";
      A     "M27_Presenza";
      R     "M42.0";
      NOP   0;
NETWORK
TITLE = PROFILATO SU RULLIERA 1 INGRESSO ESTR. LINEA 1
      A     "M42.0";
      A     "M131.1";
      S     "M27_Presenza";
      A     "M27_Presenza";
      A     "M42.3";
      R     "M27_Presenza";
      NOP   0;
NETWORK
TITLE = RICHIEDI CONFERMA TIPO BARRA SU LINEA 1
      A     "M42.0";
      FP    "M81.6";
      S     "M43.7";
      A     "Linea1_InsCoda";
      R     "M43.7";
      NOP   0;
NETWORK
TITLE = MEM PROFILATO SU RULLIERA 2 LINEA 1
      AN    "Proximity_1_pos_laser2";
      A     "M27_Presenza";
      A     "M74.4";
      S     "M42.2";
      A     "M42.2";
      A     "M42.3";
      R     "M42.2";
      NOP   0;
NETWORK
TITLE = RULLIERA 1 INGRESSO ESTR. LINEA 2 LIBERA
      A     "Proximity_1_pos_laser2";
      A     "M74.4";
      A     "M27_Presenza";
      A     "M42.2";
      =     "M42.3";
NETWORK
TITLE = MEM AUTO SOLLEVA CATENA USCITA CADENZ. LINEA 2
      AN    "M42.0";
      AN    "M27_Presenza";
      =     "M42.4";
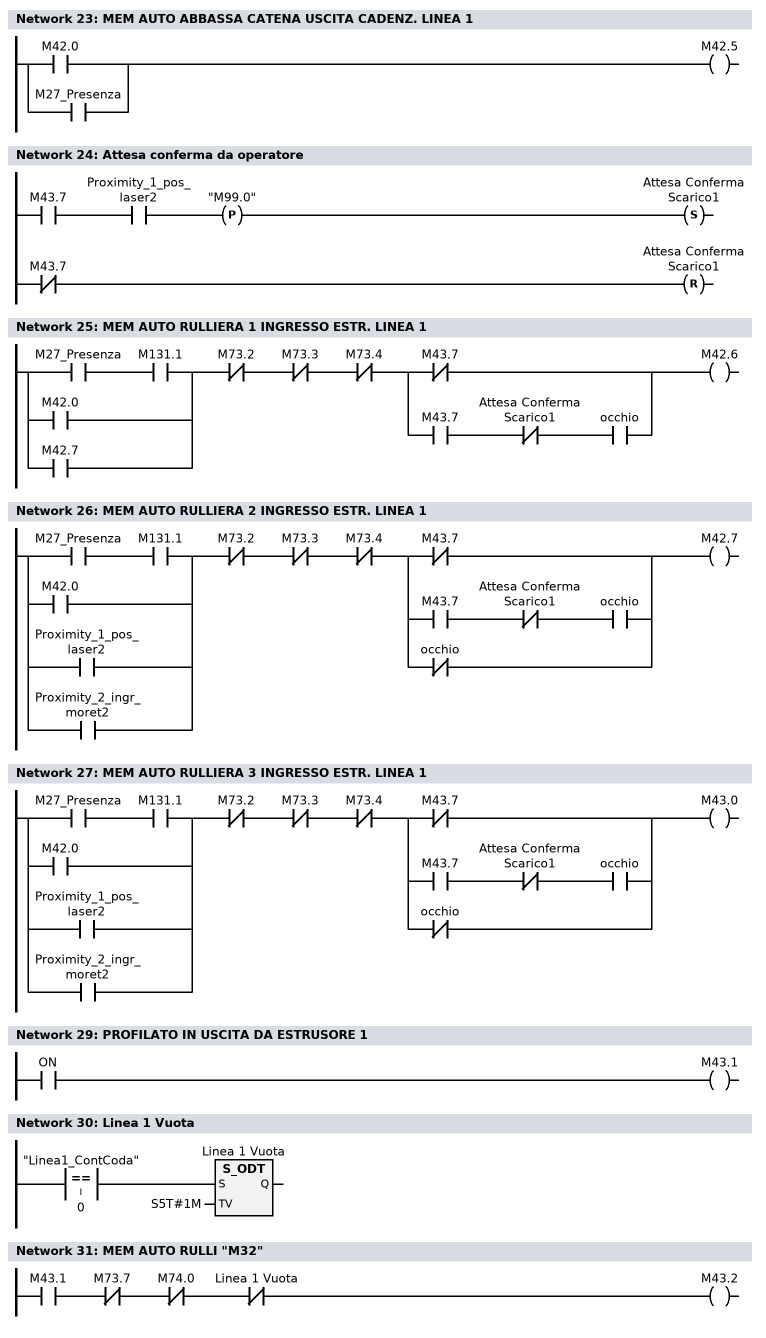
NETWORK
TITLE = MEM AUTO ABBASSA CATENA USCITA CADENZ. LINEA 1
      O     "M42.0";
      O     "M27_Presenza";
      =     "M42.5";
NETWORK
TITLE = Attesa conferma da operatore
      A     "M43.7";
      A     "Proximity_1_pos_laser2";
      FP    "M99.0";
      S     "Attesa Conferma Scarico1";
      AN    "M43.7";
      R     "Attesa Conferma Scarico1";
      NOP   0;
NETWORK
TITLE = MEM AUTO RULLIERA 1 INGRESSO ESTR. LINEA 1
      A(;
      A     "M27_Presenza";
      A     "M131.1";
      O     "M42.0";
      O     "M42.7";
      );
      AN    "M73.2";
      AN    "M73.3";
      AN    "M73.4";
      A(;
      ON    "M43.7";
      O;
      A     "M43.7";
      AN    "Attesa Conferma Scarico1";
      A     "occhio";
      );
      =     "M42.6";
NETWORK
TITLE = MEM AUTO RULLIERA 2 INGRESSO ESTR. LINEA 1
      A(;
      A     "M27_Presenza";
      A     "M131.1";
      O     "M42.0";
      O     "Proximity_1_pos_laser2";
      O     "Proximity_2_ingr_moret2";
      );
      AN    "M73.2";
      AN    "M73.3";
      AN    "M73.4";
      A(;
      ON    "M43.7";
      O;
      A     "M43.7";
      AN    "Attesa Conferma Scarico1";
      A     "occhio";
      ON    "occhio";
      );
      =     "M42.7";
NETWORK
TITLE = MEM AUTO RULLIERA 3 INGRESSO ESTR. LINEA 1
      A(;
      A     "M27_Presenza";
      A     "M131.1";
      O     "M42.0";
      O     "Proximity_1_pos_laser2";
      O     "Proximity_2_ingr_moret2";
      );
      AN    "M73.2";
      AN    "M73.3";
      AN    "M73.4";
      A(;
      ON    "M43.7";
      O;
      A     "M43.7";
      AN    "Attesa Conferma Scarico1";
      A     "occhio";
      ON    "occhio";
      );
      =     "M43.0";
NETWORK
TITLE =
NETWORK
TITLE = PROFILATO IN USCITA DA ESTRUSORE 1
      A     "ON";
      =     "M43.1";
NETWORK
TITLE = Linea 1 Vuota
      A(;
      L     "Linea1_ContCoda";
      L     0;
      ==I;
      );
      L     S5T#1M;
      SD    "Linea 1 Vuota";
      NOP   0;
      NOP   0;
      NOP   0;
      NOP   0;
NETWORK
TITLE = MEM AUTO RULLI "M32"
      A     "M43.1";
      AN    "M73.7";
      AN    "M74.0";
      AN    "Linea 1 Vuota";
      =     "M43.2";
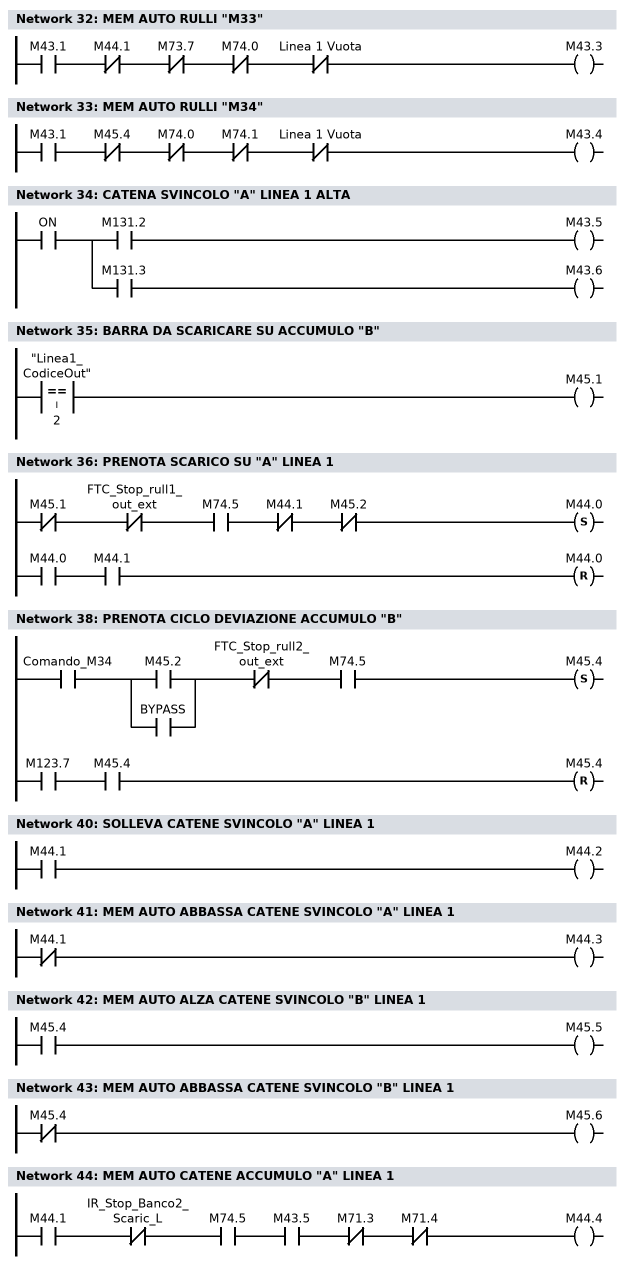
NETWORK
TITLE = MEM AUTO RULLI "M33"
      A     "M43.1";
      AN    "M44.1";
      AN    "M73.7";
      AN    "M74.0";
      AN    "Linea 1 Vuota";
      =     "M43.3";
NETWORK
TITLE = MEM AUTO RULLI "M34"
      A     "M43.1";
      AN    "M45.4";
      AN    "M74.0";
      AN    "M74.1";
      AN    "Linea 1 Vuota";
      =     "M43.4";
NETWORK
TITLE = CATENA SVINCOLO "A" LINEA 1 ALTA
      A     "ON";
      =     L 0.0;
      A     L 0.0;
      A     "M131.2";
      =     "M43.5";
      A     L 0.0;
      A     "M131.3";
      =     "M43.6";
NETWORK
TITLE = BARRA DA SCARICARE SU ACCUMULO "B"
      L     "Linea1_CodiceOut";
      L     2;
      ==I;
      =     "M45.1";
NETWORK
TITLE = PRENOTA SCARICO SU "A" LINEA 1
      AN    "M45.1";
      AN    "FTC_Stop_rull1_out_ext";
      A     "M74.5";
      AN    "M44.1";
      AN    "M45.2";
      S     "M44.0";
      A     "M44.0";
      A     "M44.1";
      R     "M44.0";
      NOP   0;
NETWORK
TITLE = SPOSTA BARRA SU RULLIERA "M34"
      A(;
      A     "M45.1";
      AN    "FTC_Stop_rull1_out_ext";
      A     "M74.5";
      AN    "M44.1";
      A     "M43.6";
      S     "M45.2";
      A     "M45.4";
      A     "M45.2";
      R     "M45.2";
      A     "M45.2";
      );
      FP    "M82.2";
      S     "Linea1_DelCoda";
NETWORK
TITLE = PRENOTA CICLO DEVIAZIONE ACCUMULO "B"
      A     "Comando_M34";
      A(;
      O     "M45.2";
      O     "BYPASS";
      );
      AN    "FTC_Stop_rull2_out_ext";
      A     "M74.5";
      S     "M45.4";
      A     "M123.7";
      A     "M45.4";
      R     "M45.4";
      NOP   0;
NETWORK
TITLE = CARICA SU SCARICO "A" LINEA 1
      A(;
      A(;
      AN    "FTC_Stop_rull1_out_ext";
      L     S5T#100MS;
      SD    "T123";
      NOP   0;
      NOP   0;
      NOP   0;
      A     "T123";
      );
      A     "Comando_M33";
      A     "M44.0";
      A     "M74.5";
      A     "M43.6";
      S     "M44.1";
      A     "M123.5";
      A     "M44.1";
      R     "M44.1";
      A     "M44.1";
      );
      FP    "M82.3";
      S     "Linea1_DelCoda";
NETWORK
TITLE = SOLLEVA CATENE SVINCOLO "A" LINEA 1
      A     "M44.1";
      =     "M44.2";
NETWORK
TITLE = MEM AUTO ABBASSA CATENE SVINCOLO "A" LINEA 1
      AN    "M44.1";
      =     "M44.3";
NETWORK
TITLE = MEM AUTO ALZA CATENE SVINCOLO "B" LINEA 1
      A     "M45.4";
      =     "M45.5";
NETWORK
TITLE = MEM AUTO ABBASSA CATENE SVINCOLO "B" LINEA 1
      AN    "M45.4";
      =     "M45.6";
NETWORK
TITLE = MEM AUTO CATENE ACCUMULO "A" LINEA 1
      A     "M44.1";
      AN    "IR_Stop_Banco2_Scaric_L";
      A     "M74.5";
      A     "M43.5";
      AN    "M71.3";
      AN    "M71.4";
      =     "M44.4";
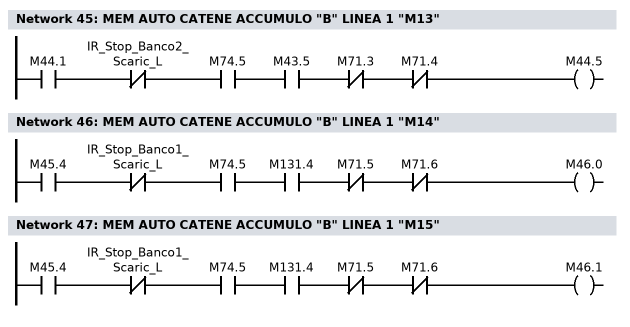
NETWORK
TITLE = MEM AUTO CATENE ACCUMULO "B" LINEA 1 "M13"
      A     "M44.1";
      AN    "IR_Stop_Banco2_Scaric_L";
      A     "M74.5";
      A     "M43.5";
      AN    "M71.3";
      AN    "M71.4";
      =     "M44.5";
NETWORK
TITLE = MEM AUTO CATENE ACCUMULO "B" LINEA 1 "M14"
      A     "M45.4";
      AN    "IR_Stop_Banco1_Scaric_L";
      A     "M74.5";
      A     "M131.4";
      AN    "M71.5";
      AN    "M71.6";
      =     "M46.0";
NETWORK
TITLE = MEM AUTO CATENE ACCUMULO "B" LINEA 1 "M15"
      A     "M45.4";
      AN    "IR_Stop_Banco1_Scaric_L";
      A     "M74.5";
      A     "M131.4";
      AN    "M71.5";
      AN    "M71.6";
      =     "M46.1";
END_FUNCTION

